// TwinCAT 3 PLC project PLC
// Title: PSAT Nell1
// Company: RMTH GmbH
// ProjectVersion: 0.1
// ProgramVersion: 3.1.4026.20
// libraries:
//   Balluff Sesnor Library TC3, * (Balluff GmbH)
//   IO Link Device Read Conditionmonitoring Data, * (Balluff GmbH)
//   IO Link Device Parametrization , * (Balluff GmbH)
//   RMTH TC3 Library, * (RMTH GmbH)
//   Tc2_ControllerToolbox, * (Beckhoff Automation GmbH)
//   Tc2_Drive, * (Beckhoff Automation GmbH)
//   Tc2_EtherCAT, * (Beckhoff Automation GmbH)
//   Tc2_IoFunctions, * (Beckhoff Automation GmbH)
//   Tc2_Math, * (Beckhoff Automation GmbH)
//   Tc2_MC2, * (Beckhoff Automation GmbH)
//   Tc2_MC2_Drive, * (Beckhoff Automation GmbH)
//   Tc2_Standard, * (Beckhoff Automation GmbH)
//   Tc2_System, * (Beckhoff Automation GmbH)
//   Tc2_TempController, * (Beckhoff Automation GmbH)
//   Tc2_Utilities, * (Beckhoff Automation GmbH)
//   Tc3_EventLogger, * (Beckhoff Automation GmbH)
//   Tc3_Module, * (Beckhoff Automation GmbH)
//   VisuDialogs, * (System)
// project tree:
//   Background/UnitTest/Enumerations/ E_TestCaseState.TcDUT, E_TestResult.TcDUT
//   Background/UnitTest/Interfaces/ ITestCase.TcIO
//   Background/UnitTest/ P_UnitTest.TcPOU
//   Background/UnitTest/TestCases/Base/ FB_TestCaseBase.TcPOU
//   Background/UnitTest/TestCases/ FB_TestCase01FileLog.TcPOU, FB_TestCase02SystemInfo.TcPOU, FB_TestCase03Station.TcPOU
//   Background/UnitTest/TestCases/StationTest/ FB_TestStation.TcPOU
//   Background/UnitTest/TestCases/StationTest/Structures/ ST_TestStation_IN.TcDUT, ST_TestStation_IO.TcDUT, ST_TestStation_OUT.TcDUT
//   DUTs/Configuration/ ST_Configuration.TcDUT
//   GVLs/ CONST.TcGVL, GVL.TcGVL, HMI.TcGVL, IO.TcGVL, NcIO.TcGVL, Safety.TcGVL, Services.TcGVL, Plant.TcGVL
//   / PlcTask.TcTTO, PlcTaskFast.TcTTO
//   POUs/Components/AxisDriver/Enumerations/ E_Axis.TcDUT, E_GearMode.TcDUT, E_JogDirection.TcDUT, E_ManualMode.TcDUT, E_MotionCommand.TcDUT, E_Mover_XTS.TcDUT, E_SoECommand.TcDUT
//   POUs/Components/AxisDriver/ FB_AxisCoupleSync2.TcPOU, FB_AxisDriver.TcPOU, FB_Axis_Ui.TcPOU
//   POUs/Components/AxisDriver/Interfaces/ ITFMotionComponent.TcIO
//   POUs/Components/AxisDriver/Structures/AdditionalAxisIO/ ST_AxisIn.TcDUT, ST_AxisIO.TcDUT, ST_AxisOut.TcDUT, ST_AxisVirtualIO.TcDUT
//   POUs/Components/AxisDriver/Structures/SoE/ ST_AxisSoE.TcDUT
//   POUs/Components/AxisDriver/Structures/ ST_AxisDriverParameter.TcDUT, ST_AxisGearInParameter.TcDUT, ST_AxisGearOutParameter.TcDUT, ST_AxisManager.TcDUT, ST_AxisTorqCtrlParameter.TcDUT, ST_AxisGeneralParameter.TcDUT, ST_AxisHaltParameter.TcDUT, ST_AxisHomingParameter.TcDUT, ST_AxisJogAccParameter.TcDUT, ST_AxisJogParameter.TcDUT, ST_AxisMoveAbsParameter.TcDUT, ST_AxisMoveAddParameter.TcDUT, ST_AxisMoveModParameter.TcDUT, ST_AxisMoveParameter.TcDUT, ST_AxisMoveRelParameter.TcDUT, ST_AxisMoveVelParameter.TcDUT, ST_AxisSetPosParameter.TcDUT, ST_AxisStopParameter.TcDUT, ST_HmiAxisManager.TcDUT
//   POUs/Components/AxisDriver/Utilities/ FB_AxisDistanceTrigger.TcPOU, FB_LimitSwitchRefSim.TcPOU, F_SpeedReached.TcPOU, F_SpeedWindowReached.TcPOU, F_TargetReached.TcPOU, F_TargetReachedOrHigher.TcPOU, F_TargetReachedOrLower.TcPOU, F_TargetWindowReached.TcPOU, F_TargetWindowReachedAxisRef.TcPOU
//   POUs/Components/CylinderDriver/ FB_Cylinder_Ui.TcPOU
//   POUs/Components/Device/ FB_Device.TcPOU, FB_Device_Ui.TcPOU
//   POUs/Components/Device/Structures/ ST_DeviceIn.TcDUT, ST_DeviceIO.TcDUT, ST_DeviceOut.TcDUT
//   POUs/Components/DriveFu/ FB_Drive.TcPOU, FB_Drive_Ui.TcPOU, FB_DriveFuAx_Ui.TcPOU
//   POUs/Components/FurnaceDriver/Enumeration/ E_FurnaceSeq.TcDUT, E_HeatingState.TcDUT
//   POUs/Components/FurnaceDriver/ FB_FurnaceDriver.TcPOU
//   POUs/Components/FurnaceDriver/Structures/ ST_FurnaceIn.TcDUT, ST_FurnaceIO.TcDUT, ST_FurnaceOut.TcDUT
//   POUs/Components/_Base/ FB_ComponentBase.TcPOU, FB_ManualUiBase.TcPOU
//   POUs/Components/_Base/Interfaces/ I_ManualUi.TcIO, ITFComponent.TcIO
//   POUs/Components/_Enumerations/ E_ComponentState.TcDUT, E_Component.TcDUT, E_ComponentType.TcDUT
//   POUs/Components/_Structures/ ST_Coordinate.TcDUT, ST_Curve.TcDUT, ST_Point.TcDUT, ST_3DPoint.TcDUT
//   POUs/HMI/Events/ FB_EventHandler.TcPOU
//   POUs/HMI/Events/Interfaces/ I_EventHandler.TcIO
//   POUs/HMI/Provider/HwHmi/ FB_HMI_PROVIDER_HW.TcPOU
//   POUs/HMI/Provider/HwHmi/Structures/+P10A_Pult/ ST_P10A_Pult_IN.TcDUT, ST_P10A_Pult_OUT.TcDUT
//   POUs/HMI/Provider/HwHmi/Structures/+P50A_Haupt/ ST_P50A_Haupt_IN.TcDUT, ST_P50A_Haupt_OUT.TcDUT
//   POUs/HMI/Provider/HwHmi/Structures/+P51A_EuchnerHandBedien/ ST_P51A_EuchnerHandB_IN.TcDUT, ST_P51A_EuchnerHandB_OUT.TcDUT
//   POUs/HMI/Provider/HwHmi/Structures/ HMI_PROVIDER_HW_IN.TcDUT, HMI_PROVIDER_HW_OUT.TcDUT, HMI_PROVIDER_HW_IO.TcDUT
//   POUs/HMI/Provider/HwHmi/Structures/_Base/ ST_PxAB_SxHandAsBs_IN.TcDUT, ST_PxAB_SxHandAsBs_OUT.TcDUT
//   POUs/HMI/Provider/Tc3Hmi/ FB_HMI_Provider_TC3.TcPOU
//   POUs/HMI/Provider/Tc3Hmi/Structures/Stations/ ST_StationToTc3Hmi.TcDUT, ST_StationFromTc3Hmi.TcDUT
//   POUs/HMI/Provider/Tc3Hmi/Structures/ ST_FromTc3Hmi.TcDUT, ST_Header.TcDUT, ST_HMI_Tc3.TcDUT, ST_ToTc3Hmi.TcDUT, ST_ToTc3HmiConditionMonitoring.TcDUT, ST_ToTc3Hmi_Door.TcDUT, ST_ToTc3Hmi_EmergencyStop.TcDUT
//   POUs/HMI/Provider/Tc3Hmi/Structures/UserControls/DataGrid/ ST_UserControlGrid_FromHmi.TcDUT, ST_UserControlGrid_ToHmi.TcDUT
//   POUs/HMI/Provider/Tc3Hmi/Structures/UserControls/ManualControl Axis/ ST_UserControl_Manual_Axis_FromHmi.TcDUT, ST_UserControl_Manual_Axis_Item.TcDUT, ST_UserControl_Manual_Axis_Item_String.TcDUT, ST_UserControl_Manual_Axis_ToHmi.TcDUT
//   POUs/HMI/Provider/Tc3Hmi/Structures/UserControls/ManualControl Cylinder/ ST_UserControl_Manual_Cylinder_FromHmi.TcDUT, ST_UserControl_Manual_Cylinder_ToHmi.TcDUT
//   POUs/HMI/Provider/Tc3Hmi/Structures/UserControls/ManualControl Device/ ST_UserControl_Manual_Device_FromHmi.TcDUT, ST_UserControl_Manual_Device_ToHmi.TcDUT
//   POUs/HMI/Provider/Tc3Hmi/Structures/UserControls/ManualControl Drive/ ST_UserControl_Manual_Drive_FromHmi.TcDUT, ST_UserControl_Manual_Drive_ToHmi.TcDUT
//   POUs/HMI/Provider/Tc3Hmi/Structures/UserControls/SensorActor/ ST_ToVisuSensorActor.TcDUT
//   POUs/HMI/Provider/_Base/ FB_HMI_PROVIDER_BASE.TcPOU
//   POUs/HMI/Provider/_Enumerations/ E_HMI_CONTROL_REQUEST.TcDUT, E_HMI_PROVIDER.TcDUT
//   POUs/HMI/Provider/_Interfaces/ ITF_HMI_PROVIDER.TcIO
//   POUs/HMI/Utilities/DynTxt/ F_CreateDynText.TcPOU, F_CreateDynTextDefault.TcPOU, F_CreateDynTextDefaultS.TcPOU, F_CreateDynTextEx.TcPOU
//   POUs/HMI/Utilities/ FB_CounterHandling.TcPOU, FB_MonitoringHandling.TcPOU, FB_ProviderRequestTrigger.TcPOU, F_AlarmPrioToText.TcPOU, F_AlarmPrioToHexColor.TcPOU, FB_HmiBaseControlTrigger.TcPOU
//   POUs/HMI/Utilities/SettingsHandling/ FB_SettingsHandling.TcPOU, F_SettingItemHandling.TcPOU, F_SettingItemHandlingB.TcPOU, F_SettingItemHandlingF.TcPOU, F_SettingItemHandlingI.TcPOU, F_SettingItemHandlingWs.TcPOU
//   POUs/HMI/Utilities/Tracking/ F_TrackSettingChangesB.TcPOU, F_TrackSettingChangesF.TcPOU, F_TrackSettingChangesI.TcPOU, F_TrackSettingChangesT.TcPOU, F_TrackSettingChangesWs.TcPOU
//   POUs/HMI/Utilities/Validation/ F_ChkSettingLimit.TcPOU, F_ChkSettingLimitF.TcPOU, F_ChkSettingLimitN.TcPOU, F_ChkSettingUserLevel.TcPOU
//   POUs/HMI/ P_HMI_Controller.TcPOU
//   POUs/HMI/_Enumerations/ E_Axis_JogMode.TcTLEO, E_DataType.TcTLEO, E_Drive_JogMode.TcDUT, E_Language.TcDUT, E_ManualObjectControlMode.TcDUT, E_Popup.TcDUT, E_RecipeMode.TcTLEO, E_User.TcTLEO, E_User_Level.TcDUT
//   POUs/HMI/_Structures/Counter/ E_CounterReaction.TcTLEO, ST_CounterControlIn.TcDUT, ST_CounterControlOut.TcDUT, ST_Counter_Item_String.TcDUT
//   POUs/HMI/_Structures/Data/ ST_Data_Item_String.TcDUT, ST_Data_Item.TcDUT
//   POUs/HMI/_Structures/Monitoring/ ST_GridObject_Name_Value1_Event1_Value2_Event2_Unit.TcDUT, ST_GridObject_Name_sValue_Unit.TcDUT, ST_Monitoring_Station.TcDUT, ST_Monitoring.TcDUT, ST_Monitoring_Base.TcDUT, ST_Monitoring_Module.TcDUT
//   POUs/HMI/_Structures/Popup/ E_PopupSymbol.TcDUT, ST_PopUp_FromHmi.TcDUT, ST_PopUp_ToHmi.TcDUT
//   POUs/HMI/_Structures/Recipe/ ST_HMI_RECIPE_IN.TcDUT, ST_HMI_RECIPE_OUT.TcDUT
//   POUs/HMI/_Structures/Safety/ ST_HMI_SAFETY_IN.TcDUT, ST_HMI_SAFETY_OUT.TcDUT
//   POUs/HMI/_Structures/Settngs/ ST_HMI_CONTROL_SETTING_IN.TcDUT, ST_HMI_CONTROL_SETTING_OUT.TcDUT, ST_HMI_CONTROL_SETTING_STATION_OUT.TcDUT, ST_HMI_CONTROL_SETTING_MODULE_OUT.TcDUT, ST_HMI_CONTROL_SETTING_ITEM_IN.TcDUT, ST_HMI_CONTROL_SETTING_ITEM_OUT.TcDUT
//   POUs/HMI/_Structures/SetupPlant/ E_SetupPlantShape.TcDUT, E_SetupPlantStateShape.TcDUT, ST_SetupPlant_Item_String.TcDUT
//   POUs/HMI/_Structures/ ST_HMI.TcDUT, ST_HMI_IN.TcDUT, ST_HMI_InOut.TcDUT, ST_HMI_OUT.TcDUT, ST_NameValue.TcDUT
//   POUs/HMI/_Structures/UserManagment/ ST_HMI_USER_MGMT_IN.TcDUT, ST_HMI_USER_MGMT_OUT.TcDUT, ST_User_Management.TcDUT
//   POUs/HMI/_Structures/_Base/Button/ ST_HMI_BUTTON_IN.TcDUT, ST_HMI_BUTTON_OUT.TcDUT
//   POUs/HMI/_Structures/_Base/Common/ ST_HMI_BASE_CONTROL_IN.TcDUT, ST_HMI_BASE_CONTROL_OUT.TcDUT, ST_HMI_BASE_SPECIAL_IN.TcDUT, ST_HMI_GRID_IN.TcDUT, ST_HMI_NAME_VALUE_STRING.TcDUT, ST_HMI_TRAFFIC_LIGHT_OUT.TcDUT
//   POUs/HMI/_Structures/_Base/Manual/ManualControl Axis/ ST_HMI_MANUAL_AXIS_IN.TcDUT, ST_HMI_MANUAL_AXIS_ITEM.TcDUT, ST_HMI_MANUAL_AXIS_ITEM_STRING.TcDUT, ST_HMI_MANUAL_AXIS_OUT.TcDUT
//   POUs/HMI/_Structures/_Base/Manual/ManualControl Cylinder/ ST_HMI_MANUAL_CYLINDER_IN.TcDUT, ST_HMI_MANUAL_CYLINDER_OUT.TcDUT
//   POUs/HMI/_Structures/_Base/Manual/ManualControl Device/ ST_HMI_MANUAL_DEVICE_IN.TcDUT, ST_HMI_MANUAL_DEVICE_OUT.TcDUT
//   POUs/HMI/_Structures/_Base/Manual/ManualControl Drive/ ST_HMI_MANUAL_DRIVE_IN.TcDUT, ST_HMI_MANUAL_DRIVE_OUT.TcDUT
//   POUs/HMI/_Structures/_Base/Module/ ST_HMI_BASE_MODULE_IN.TcDUT, ST_HMI_BASE_MODULE_MANUAL_IN.TcDUT, ST_HMI_BASE_MODULE_MANUAL_OUT.TcDUT, ST_HMI_BASE_MODULE_OUT.TcDUT
//   POUs/HMI/_Structures/_Base/Station/ ST_HMI_BASE_STATION_IN.TcDUT, ST_HMI_BASE_STATION_MANUAL_IN.TcDUT, ST_HMI_BASE_STATION_MANUAL_OUT.TcDUT, ST_HMI_BASE_STATION_OUT.TcDUT
//   POUs/HMI/_Structures/_Base/ ST_HMI_BASE_IN.TcDUT, ST_HMI_BASE_OUT.TcDUT
//   POUs/HMI/_Structures/_Common/ ST_HexColor.TcDUT, ST_HMI_COLOR_STRING.TcDUT, ST_Text.TcDUT, ST_DefaultHmiToPlc.TcDUT
//   POUs/HMI/_Structures/_TextLists/ ST_Text_List_Components.TcDUT, ST_Text_List_Global.TcDUT, ST_Text_List_Safety.TcDUT, ST_Text_List_System.TcDUT
//   POUs/Items/TcaCarrier/Enumerations/ eTcaCarrierCmd.TcDUT, eTcaCarrierLayout.TcDUT
//   POUs/Items/TcaCarrier/Structures/ TcaCarrierConfig.TcDUT, TcaCarrierData.TcDUT, TcaCarrierService.TcDUT
//   POUs/Items/TcaCarrier/ TcaCarrier.TcPOU
//   POUs/Items/TcaTrolley/Structures/ TcaTrolleyConfig.TcDUT, TcaTrolleyData.TcDUT, TcaTrolleyService.TcDUT
//   POUs/Items/TcaTrolley/ TcaTrolley.TcPOU
//   POUs/Items/TcaWorkpiece/Enumerations/ eTcaWorkpieceShape.TcDUT, eTcaWorkpieceStatus.TcDUT
//   POUs/Items/TcaWorkpiece/Structures/ TcaWorkpieceData.TcDUT
//   POUs/Items/TcaWorkpiece/ TcaWorkpieceControl.TcPOU
//   POUs/ MAIN.TcPOU, MAIN_Fast.TcPOU
//   POUs/Plant/_Enumerations/ E_Module.TcDUT, E_PlantSettings.TcDUT, E_ProductionSettings.TcDUT, E_ProductSettings.TcDUT, E_Station.TcDUT
//   POUs/Plant/M001_Module/_Enumerations/ E_M001_Settings.TcDUT
//   POUs/Plant/M001_Module/_Structures/ ST_M001_HMI_IN.TcDUT, ST_M001_Interface.TcDUT, ST_M001_HMI_OUT.TcDUT, ST_M001_IO.TcDUT, ST_M001_IO_IN.TcDUT, ST_M001_IO_OUT.TcDUT
//   POUs/Plant/ P_Plant.TcPOU
//   POUs/Plant/ST010_OvenA/_Structures/ ST_St010_HMI_IN.TcDUT, ST_St010_Interface.TcDUT, ST_St010_HMI_IN_OUT.TcDUT, ST_St010_HMI_OUT.TcDUT, ST_St010_IO_IN.TcDUT, ST_St010_IO.TcDUT, ST_St010_IO_OUT.TcDUT
//   POUs/Plant/ST020_OvenB/_Enumerations/ E_St020_Settings.TcDUT
//   POUs/Plant/ST020_OvenB/ FB_St020_OvenB.TcPOU
//   POUs/Plant/ST020_OvenB/_Structures/ ST_St020_HMI_IN_OUT.TcDUT, ST_St020_HMI_IN.TcDUT, ST_St020_Interface.TcDUT, ST_St020_IO.TcDUT, ST_St020_IO_IN.TcDUT, ST_St020_IO_OUT.TcDUT, ST_St020_HMI_OUT.TcDUT
//   POUs/Plant/ST030_Handling/_Enumerations/ E_St030_Command.TcDUT, E_St030_EmptySlotChk.TcDUT, E_St030_Settings.TcDUT
//   POUs/Plant/ST030_Handling/ FB_St030_Handling.TcPOU
//   POUs/Plant/ST030_Handling/_Structures/ ST_St030_HMI_OUT.TcDUT, ST_St030_HMI_IN.TcDUT, ST_St030_Interface.TcDUT, ST_St030_Command.TcDUT, ST_St030_IO.TcDUT, ST_St030_IO_IN.TcDUT, ST_St030_IO_OUT.TcDUT, ST_St030_HMI_IN_OUT.TcDUT, ST_XZ_Point.TcDUT
//   POUs/Plant/ST040_Storage/_Enumerations/ E_St040_Settings.TcDUT
//   POUs/Plant/ST040_Storage/ FB_St040_Storage.TcPOU
//   POUs/Plant/ST040_Storage/_Structures/ ST_St040_HMI_IN.TcDUT, ST_St040_HMI_IN_OUT.TcDUT, ST_St040_HMI_OUT.TcDUT, ST_St040_IO.TcDUT, ST_St040_IO_IN.TcDUT, ST_St040_IO_OUT.TcDUT, ST_St040_Interface.TcDUT
//   POUs/Plant/ST050_Mould/_Enumerations/ E_St050_Settings.TcDUT
//   POUs/Plant/ST050_Mould/ FB_St050_Mould.TcPOU
//   POUs/Plant/ST050_Mould/_Structures/ ST_St050_Interface.TcDUT, ST_St050_IO.TcDUT, ST_St050_IO_IN.TcDUT, ST_St050_IO_OUT.TcDUT, TcaEngelCastingCarrierInput.TcDUT, TcaEngelCastingCarrierJob.TcDUT, TcaEngelCastingCarrierJobStatus.TcDUT, TcaEngelCastingCarrierOutput.TcDUT, TcaEngelCastingCarrierStatus.TcDUT
//   POUs/Plant/_Base/Interfaces/ IModule.TcIO, IStation.TcIO
//   POUs/Plant/_Specific/Components/TcaWorkpiece/ TcaWorkpieceControl.TcPOU (not stored)
//   POUs/Plant/_Specific/S01_Workpiece/Enumerations/ E_HMI_WP_CMD.TcDUT (not stored), E_ProcessState.TcDUT (not stored), E_ProcessStep.TcDUT (not stored)
//   POUs/Plant/_Specific/S01_Workpiece/ FB_Workpiece.TcPOU (not stored), FB_WorkpieceRef.TcPOU (not stored)
//   POUs/Plant/_Specific/S01_Workpiece/Structures/ ST_HMI_WP_CMD.TcDUT (not stored), ST_Workpiece.TcDUT (not stored)
//   POUs/Plant/_Specific/S02_Pallet/Enumerations/ E_HMI_PL_CMD.TcDUT (not stored)
//   POUs/Plant/_Specific/S02_Pallet/ FB_Pallet.TcPOU (not stored), FB_PalletRef.TcPOU (not stored)
//   POUs/Plant/_Specific/S02_Pallet/Structures/ ST_HMI_PL_CMD.TcDUT (not stored), ST_Pallet.TcDUT (not stored)
//   POUs/Plant/_Specific/S03_Trolley/Enumerations/ E_HMI_TR_CMD.TcDUT (not stored)
//   POUs/Plant/_Specific/S03_Trolley/ FB_Trolley.TcPOU (not stored)
//   POUs/Plant/_Specific/S03_Trolley/Structures/ ST_HMI_TR_CMD.TcDUT (not stored), ST_Trolley.TcDUT (not stored)
//   POUs/Plant/_Structures/ControlCabinet/ ST_ControlCabinetIn.TcDUT, ST_ControlCabinetIO.TcDUT, ST_ControlCabinetOut.TcDUT
//   POUs/Plant/_Structures/Counter/ ST_Counter.TcDUT
//   POUs/Plant/_Structures/Objects/ ST_Objects.TcDUT, ST_Object_Item.TcDUT
//   POUs/Plant/_Structures/Settings/ ST_ModuleDynSettings.TcDUT, ST_Settings.TcDUT, ST_StationDynSettings.TcDUT
//   POUs/Plant/_Structures/ ST_DefaultEventClasses.TcDUT, ST_MODULE_STATIONS_INFO.TcDUT, ST_MODULES_INFO.TcDUT
//   POUs/Safety/Components/Euchner_MBM/ FB_Euchner_MBM.TcPOU
//   POUs/Safety/Components/Euchner_MBM/Structure/ ST_Euchner_MBM_HW_IN.TcDUT, ST_Euchner_MBM_HW_OUT.TcDUT, ST_Euchner_MBM_IN.TcDUT, ST_Euchner_MBM_OUT.TcDUT, ST_MBM_IO.TcDUT
//   POUs/Safety/Components/Euchner_MGB2/ FB_SafeDoorMGB2.TcPOU
//   POUs/Safety/Components/Euchner_MGB2/Structure/MGB2/ ST_Euchner_MGB2_HW_IN.TcDUT, ST_Euchner_MGB2_HW_OUT.TcDUT, ST_Euchner_MGB2_IN.TcDUT, ST_Euchner_MGB2_OUT.TcDUT
//   POUs/Safety/Components/Euchner_MGB2/Structure/MSM/ ST_Euchner_MSM_DA_IN.TcDUT, ST_Euchner_MSM_DA_OUT.TcDUT, ST_Euchner_MSM_HW_IN.TcDUT, ST_Euchner_MSM_HW_OUT.TcDUT, ST_Euchner_MSM_IN.TcDUT, ST_Euchner_MSM_OUT.TcDUT
//   POUs/Safety/Components/Euchner_MGB2/Structure/ ST_MGB2_IO.TcDUT
//   POUs/Safety/Components/SafetyDoor/ FB_SafetyDoor.TcPOU
//   POUs/Safety/Components/SafetyDoor/Structure/ ST_SafetyDoor_IN.TcDUT, ST_SafetyDoor_IO.TcDUT, ST_SafetyDoor_OUT.TcDUT
//   POUs/Safety/Enumerations/ E_EDM_Out.TcDUT, E_Safety_Actor.TcDUT, E_EmergencyStop.TcDUT, E_Door.TcDUT
//   POUs/Safety/ P_Safety.TcPOU
//   POUs/Safety/Structures/Diag/ E_HistoryDiagDevices.TcDUT, ST_DiagHistory.TcDUT, ST_DiagMessage.TcDUT, ST_DiagMessageFlags.TcDUT, ST_ELM3xxxPAIInfoData.TcDUT, ST_MessageItem.TcDUT, ST_SafetyDiagInfo.TcDUT
//   POUs/Safety/Structures/ ST_SafetyIn.TcDUT, ST_SafetyIO.TcDUT, ST_SafetyOut.TcDUT
//   POUs/Safety/TwinSAFE_Diagnose/ FB_Diagnosis_History.TcPOU, FB_TwinSAFEDiag_EDM.TcPOU, FB_TwinSAFEDiag_EmergencyStop.TcPOU, FB_TwinSAFEDiag_MachineMonitoring.TcPOU, FB_TwinSAFEDiag_TwoHand.TcPOU, FB_TwinSAFE_HW_Diag.TcPOU
//   POUs/Plant/M001_Module/ FB_M001_Module.TcPOU
//   POUs/Plant/ST010_OvenA/_Enumerations/ E_St010_Settings.TcDUT
//   POUs/Plant/_Base/ FB_ModuleBase.TcPOU, FB_StationBase.TcPOU
//   POUs/Plant/ST010_OvenA/ FB_St010_OvenA.TcPOU
//   POUs/System/ P_SysSrv.TcPOU
//   POUs/System/Recipe/ FB_RecipeManager.TcPOU
//   POUs/System/Supervision/Enumerations/Alarmsystem/ E_AlarmPriority.TcDUT, E_AlarmState.TcDUT, E_EventReaction.TcDUT
//   POUs/System/Supervision/Enumerations/ E_EtherCatBox.TcDUT
//   POUs/System/Supervision/EtherCAT/Enumerations/ E_EcDeviceState.TcDUT
//   POUs/System/Supervision/EtherCAT/ FB_DiagEtherCAT.TcPOU
//   POUs/System/Supervision/ImplicitChecks/ CheckBounds.TcPOU, CheckDivDInt.TcPOU, CheckDivLInt.TcPOU, CheckDivLReal.TcPOU, CheckDivReal.TcPOU, CheckPointer.TcPOU, CheckRangeSigned.TcPOU, CheckRangeUnsigned.TcPOU
//   POUs/System/Supervision/ P_Supervision.TcPOU
//   POUs/System/Supervision/Structures/ ST_EcMaster_In.TcDUT, ST_GridObject_Register.TcDUT, ST_SystemVars.TcDUT
//   POUs/System/Utilities/Convert/ F_DegPerSecToDegPerMin.TcPOU, F_DegPerSecToUpm.TcPOU, F_Diagnostic_EcDeviceState.TcPOU, F_Diagnostic_EcLinkState.TcPOU, F_Diagnostic_EcMasterDeviceState.TcPOU, F_EcDeviceTimeStampToTime.TcPOU, F_MeterPerMinToMmPerSec.TcPOU, F_MmPerSecToMmPerMin.TcPOU, F_UpmToDegreePerSec.TcPOU, F_MmPerMinToMmPerSec.TcPOU, F_MmPerSecToMeterPerMin.TcPOU, F_DegPerMinToDegPerSec.TcPOU
//   POUs/System/Utilities/Counter/ E_Counter.TcDUT, E_CounterMode.TcDUT, F_Counter.TcPOU, ST_Counter_Item.TcDUT
//   POUs/System/Utilities/CSV/ FB_WriteCSV.TcPOU
//   POUs/System/Utilities/CSV/Structures/ ST_FillOrder.TcDUT
//   POUs/System/Utilities/ FB_JogTrigTon.TcPOU, FB_Puls_On_Off.TcPOU, FB_RtrigFtrigTof.TcPOU, FB_RtrigFtrig.TcPOU, FB_StableValue.TcPOU, FB_ToggleSwitch.TcPOU
//   POUs/System/Utilities/Functions/ F_ADD_REF_F.TcPOU, F_AND_REF_EX.TcPOU, F_Byte_To_DWord.TcPOU, F_Byte_To_Word.TcPOU, F_ColorToStringHexColor.TcPOU, F_CutInstancePath.TcPOU, F_FindBackupItem.TcPOU, F_FormatString.TcPOU, F_InitDynDataItem.TcPOU, F_InRange.TcPOU, F_Log_Add.TcPOU, F_OR_REF.TcPOU, F_AND_REF.TcPOU, F_OR_REF_EX.TcPOU, F_Real_To_Byte.TcPOU, F_RestoreSettingValues.TcPOU, F_Settings_Management.TcPOU, F_Settings_Row_Delete.TcPOU, F_Settings_Row_Insert.TcPOU, F_Trend.TcPOU, F_CopyDataItemValues.TcPOU
//   POUs/System/Utilities/Interfaces/ I_StringBuilder.TcIO, I_WStringBuilder.TcIO
//   POUs/System/Utilities/Sequencer/ FB_SequenceHelper.TcPOU, FB_SequenceHelperSb.TcPOU
//   POUs/System/Utilities/String/ FB_StringBuilder.TcPOU, FB_WStringBuilder.TcPOU, F_Replace.TcPOU, WConcat10.TcPOU, WConcat2x.TcPOU, WConcat3.TcPOU, WConcat4.TcPOU, WConcat5.TcPOU, WConcat6.TcPOU, WConcat7.TcPOU, WConcat8.TcPOU, WConcat9.TcPOU
//   POUs/System/Utilities/Var2File/ FB_Var2File.TcPOU
//   POUs/System/Utilities/Var2File/Structures/ ST_Var2File_Com.TcDUT, ST_Var2File_Config.TcDUT
// real-time tasks:
//   TASK PlcTask: cycle T#5ms, priority 10, ADS port 350
//   TASK PlcTaskFast: cycle T#1ms, priority 4, ADS port 351
// motion (NC):
//   TASK NC-Task 1 SAF: cycle T#2ms, priority 6, ADS port 501
//   TASK NC-Task 1 SVB: cycle T#10ms, priority 12, ADS port 511
//   AXIS Oven B CH1 (id 14)
//     Dynamic: Acceleration=282800000, Deceleration=282800000, Jerk=2.85628e+17
//     Velo: RefSearch=25, RefSync=25, SlowManual=14, FastManual=28, Maximum=28
//     PositionAreaControl: Enable=false
//     TargetPosControl: Enable=false
//     OtherSettings: AllowMotionCmdToSlave=true
//     encoder EncType=7
//       EncPara: ScaleFactorNumerator=0.001879, Offset=-1.4, MaxCount=#x0000ffff, ReferenceSystem=1
//     drive DrvType=23
//       Analog: VeloReferenz=28, TorqueSetpointScale=10, ScaleFactorActTorque=0.1
//       TimeComp: TaskDelayCycles=1
//     controller CtrType=1
//       CtrPara: PriorControlFactor=1
//         PosDiffControl: Enable=false
//         Observer: BandWidth=20
//   AXIS Oven B CH2 (id 15)
//     Dynamic: Acceleration=282800000, Deceleration=282800000, Jerk=2.85628e+17
//     Velo: RefSearch=25, RefSync=25, SlowManual=14, FastManual=28, Maximum=28
//     PositionAreaControl: Enable=false
//     TargetPosControl: Enable=false
//     OtherSettings: AllowMotionCmdToSlave=true
//     encoder EncType=7
//       EncPara: ScaleFactorNumerator=0.001879, Offset=-1.4, MaxCount=#x0000ffff, ReferenceSystem=1
//     drive DrvType=23
//       Analog: VeloReferenz=28, TorqueSetpointScale=10, ScaleFactorActTorque=0.1
//       TimeComp: TaskDelayCycles=1
//     controller CtrType=1
//       CtrPara: PriorControlFactor=1
//         PosDiffControl: Enable=false
//         Observer: BandWidth=20
//   AXIS Rackfeeder X (id 16)
//     Dynamic: AccelerationMaximum=5000, DecelerationMaximum=5000, Acceleration=2150.09, Deceleration=2150.09, Jerk=9085.86
//     Velo: RefSearch=16.41285, RefSync=16.41285, SlowManual=10, FastManual=60, Fast=1641.285, Maximum=1641.29
//     OtherSettings: AllowMotionCmdToSlave=true
//     encoder EncType=8
//       EncPara: ScaleFactorNumerator=150, ScaleFactorDenominator=10485760, MaxCount=#xffffffff, EncPositionSource=1
//     drive DrvType=9
//       DrvPara: MaxCount=#xffffffff, DriveControlDWord=#x00030100
//         Analog: VeloReferenz=1805.4135, VeloScale=1.02400649589962, TorqueSetpointScale=10, ScaleFactorActTorque=0.1
//         TimeComp: TaskDelayCycles=1
//     controller CtrType=1
//       CtrPara: PriorControlFactor=1
//         Observer: BandWidth=20
//   AXIS Rackfeeder Y (id 17)
//     Dynamic: Acceleration=2004.51, Deceleration=2004.51, Jerk=8036.12
//     Velo: RefSearch=15.04511, RefSync=15.04511, SlowManual=10, FastManual=60, Fast=1504.511, Maximum=1504.51
//     OtherSettings: AllowMotionCmdToSlave=true
//     encoder EncType=8
//       EncPara: ScaleFactorNumerator=220, ScaleFactorDenominator=16777216, MaxCount=#xffffffff, EncPositionSource=1
//     drive DrvType=9
//       DrvPara: MaxCount=#xffffffff, DriveControlDWord=#x00030100
//         Analog: VeloReferenz=1654.9621, VeloScale=1.02400649589962, TorqueSetpointScale=10, ScaleFactorActTorque=0.1
//         TimeComp: TaskDelayCycles=1
//     controller CtrType=1
//       CtrPara: PriorControlFactor=1
//         Observer: BandWidth=20
//   AXIS Rackfeeder Z (id 18)
//     Dynamic: Acceleration=500, Deceleration=500, Jerk=500
//     Velo: RefSearch=30.19555, RefSync=30.19555, SlowManual=35, FastManual=210, Fast=3019.555, Maximum=3019.555
//     OtherSettings: AllowMotionCmdToSlave=true
//     encoder EncType=8
//       EncPara: ScaleFactorNumerator=27.59625, ScaleFactorDenominator=1048576, MaxCount=#xffffffff, EncPositionSource=1
//     drive DrvType=9
//       DrvPara: MaxCount=#xffffffff, DriveControlDWord=#x00030100
//         Analog: VeloReferenz=3321.5105, VeloScale=1.02400649589962, TorqueSetpointScale=10, ScaleFactorActTorque=0.1
//         TimeComp: TaskDelayCycles=1
//     controller CtrType=1
//       CtrPara: PriorControlFactor=1
//         Observer: BandWidth=20
//   AXIS Oven B (id 21)
//     Dynamic: Acceleration=1231.0125, Deceleration=1231.0125, Jerk=3693.0375
//     Velo: RefSearch=8.20675, RefSync=8.20675, SlowManual=20, FastManual=120, Fast=820.675, Maximum=820.675
//     OtherSettings: AllowMotionCmdToSlave=true
//     encoder EncType=8
//       EncPara: ScaleFactorNumerator=120, ScaleFactorDenominator=16777216, Inverse=true, MaxCount=#xffffffff, EncPositionSource=1
//     drive DrvType=9
//       DrvPara: Inverse=true, MaxCount=#xffffffff, DriveControlDWord=#x00030100
//         Analog: VeloReferenz=902.7425, VeloScale=1.02400649589962, TorqueSetpointScale=10, ScaleFactorActTorque=0.1
//         TimeComp: TaskDelayCycles=1
//     controller CtrType=1
//       CtrPara: PriorControlFactor=1
//         Observer: BandWidth=20
//   AXIS Oven A (id 20)
//     Dynamic: Acceleration=1231.01, Deceleration=1231.01, Jerk=3693.04
//     Velo: RefSearch=8.20675, RefSync=8.20675, SlowManual=20, FastManual=120, Fast=820.675, Maximum=820.675
//     OtherSettings: AllowMotionCmdToSlave=true
//     encoder EncType=8
//       EncPara: ScaleFactorNumerator=120, ScaleFactorDenominator=16777216, Inverse=true, MaxCount=#xffffffff, EncPositionSource=1
//     drive DrvType=9
//       DrvPara: Inverse=true, MaxCount=#xffffffff, DriveControlDWord=#x00030100
//         Analog: VeloReferenz=902.7425, VeloScale=1.02400649589962, TorqueSetpointScale=10, ScaleFactorActTorque=0.1
//         TimeComp: TaskDelayCycles=1
//     controller CtrType=1
//       CtrPara: PriorControlFactor=1
//         Observer: BandWidth=20
//   AXIS Oven A CH1 (id 1)
//     Dynamic: Acceleration=282800000, Deceleration=282800000, Jerk=2.85628e+17, DelayTime=0.01, OverrideType=4
//     Velo: RefSearch=25, RefSync=25, SlowManual=14, FastManual=28, Maximum=28
//     PositionAreaControl: Enable=false
//     TargetPosControl: Enable=false
//     OtherSettings: AllowMotionCmdToSlave=true
//     encoder EncType=7
//       EncPara: ScaleFactorNumerator=0.001879, Offset=-1.4, EncMode=1, MaxCount=#x0000ffff, ReferenceSystem=1
//         FilterTime: TVelo=0.1
//         SoftEndMinControl: Range=-5
//         SoftEndMaxControl: Range=30
//         ActPosCorrection: Enable=true, Time=1
//     drive DrvType=23
//       Analog: VeloReferenz=28, TorqueSetpointScale=10, ScaleFactorActTorque=0.1
//       TimeComp: TaskDelayCycles=1
//     controller CtrType=1
//       CtrPara: PriorControlFactor=1
//         PosDiffControl: Enable=false
//         Observer: BandWidth=20
//   AXIS Oven A CH2 (id 13)
//     Dynamic: Acceleration=282800000, Deceleration=282800000, Jerk=2.85628e+17
//     Velo: RefSearch=25, RefSync=25, SlowManual=14, FastManual=28, Maximum=28
//     PositionAreaControl: Enable=false
//     TargetPosControl: Enable=false
//     OtherSettings: AllowMotionCmdToSlave=true
//     encoder EncType=7
//       EncPara: ScaleFactorNumerator=0.001879, Offset=-1.4, MaxCount=#x0000ffff, ReferenceSystem=1
//     drive DrvType=23
//       Analog: VeloReferenz=28, TorqueSetpointScale=10, ScaleFactorActTorque=0.1
//       TimeComp: TaskDelayCycles=1
//     controller CtrType=1
//       CtrPara: PriorControlFactor=1
//         PosDiffControl: Enable=false
//         Observer: BandWidth=20
//   AXIS Storage A (id 2)
//     Dynamic: Acceleration=282800000, Deceleration=282800000, Jerk=2.85628e+17, DelayTime=0.01, OverrideType=4
//     Velo: RefSearch=25, RefSync=25, SlowManual=14, FastManual=28, Maximum=28
//     PositionAreaControl: Enable=false
//     TargetPosControl: Enable=false
//     OtherSettings: AllowMotionCmdToSlave=true
//     encoder EncType=7
//       EncPara: ScaleFactorNumerator=0.001879, Offset=-1.4, EncMode=1, MaxCount=#x0000ffff, ReferenceSystem=1
//         FilterTime: TVelo=0.1
//         SoftEndMinControl: Range=-5
//         SoftEndMaxControl: Range=30
//         ActPosCorrection: Enable=true, Time=1
//     drive DrvType=23
//       Analog: VeloReferenz=28, TorqueSetpointScale=10, ScaleFactorActTorque=0.1
//       TimeComp: TaskDelayCycles=1
//     controller CtrType=1
//       CtrPara: PriorControlFactor=1
//         PosDiffControl: Enable=false
//         Observer: BandWidth=20
//   AXIS Storage B (id 3)
//     Dynamic: Acceleration=282800000, Deceleration=282800000, Jerk=2.85628e+17
//     Velo: RefSearch=25, RefSync=25, SlowManual=14, FastManual=28, Maximum=28
//     PositionAreaControl: Enable=false
//     TargetPosControl: Enable=false
//     OtherSettings: AllowMotionCmdToSlave=true
//     encoder EncType=7
//       EncPara: ScaleFactorNumerator=0.001879, Offset=-1.4, MaxCount=#x0000ffff, ReferenceSystem=1
//     drive DrvType=23
//       Analog: VeloReferenz=28, TorqueSetpointScale=10, ScaleFactorActTorque=0.1
//       TimeComp: TaskDelayCycles=1
//     controller CtrType=1
//       CtrPara: PriorControlFactor=1
//         PosDiffControl: Enable=false
//         Observer: BandWidth=20
// I/O:
//   DEVICE Gerät 3 (EtherCAT), AmsNetId 172.31.31.4.4.1
//     Klemme 1 (EK1100) [EK1100 EtherCAT-Koppler (2A E-Bus)]
//       Klemme 33 (EL6910) [EL6910, TwinSAFE PLC]
//       Klemme 3 (EL1904) [EL1904, 4 K. Safety Eingang 24V, TwinSAFE]
//         modules: Module 1 (FSOES)
//       Klemme 4 (EL2904) [EL2904, 4 K. Safety Ausgang 24V, 0.5A, TwinSAFE]
//         modules: Module 1 (FSOES), Module 2 (DO)
//       Klemme 5 (EL1104) [EL1104 4K. Dig. Eingang 24V, 3ms, Sensorversorgung]
//       Klemme 6 (EL1104) [EL1104 4K. Dig. Eingang 24V, 3ms, Sensorversorgung]
//       Klemme 7 (EL6224) [EL6224 (IO Link Master)]
//       ENGEL Interface (EL1008) [EL1008 8K. Dig. Eingang 24V, 3ms]
//       ENGEL Interface (EL2624) [EL2624 4K. Relais Ausgang, Schließer (125V AC / 30V DC)]
//       Klemme 43 (EL1904)
//       Ovens (EK1122) [EK1122 2-Port EtherCAT-Abzweig]
//         Oven_A (EK1100) [EK1100 EtherCAT-Koppler (2A E-Bus)]
//           Klemme 10 (EL1904) [EL1904, 4 K. Safety Eingang 24V, TwinSAFE]
//             modules: Module 1 (FSOES)
//           Klemme 11 (EL2904) [EL2904, 4 K. Safety Ausgang 24V, 0.5A, TwinSAFE]
//             modules: Module 1 (FSOES), Module 2 (DO)
//           Klemme 12 (EL7332) [EL7332 2K. DC-Motor-Endstufe (24V, 1.5A)]
//           Klemme 13 (EL3062-0030) [EL3062-0030 2K.Ana. Eingang 0-30V]
//           Klemme 14 (EL1004) [EL1004 4K. Dig. Eingang 24V, 3ms]
//           Klemme 15 (EL2004) [EL2004 4K. Dig. Ausgang 24V, 0.5A]
//           Klemme 51 (EL1104)
//           Klemme 16 (EL9010) [EL9010 Endklemme]
//         Oven_B (EK1100) [EK1100 EtherCAT-Koppler (2A E-Bus)]
//           Klemme 18 (EL1904) [EL1904, 4 K. Safety Eingang 24V, TwinSAFE]
//             modules: Module 1 (FSOES)
//           Klemme 19 (EL2904) [EL2904, 4 K. Safety Ausgang 24V, 0.5A, TwinSAFE]
//             modules: Module 1 (FSOES), Module 2 (DO)
//           Klemme 20 (EL7332) [EL7332 2K. DC-Motor-Endstufe (24V, 1.5A)]
//           Klemme 21 (EL3062-0030) [EL3062-0030 2K.Ana. Eingang 0-30V]
//           Klemme 22 (EL1004) [EL1004 4K. Dig. Eingang 24V, 3ms]
//           Klemme 23 (EL2004) [EL2004 4K. Dig. Ausgang 24V, 0.5A]
//           Klemme 66 (EL1104)
//           Klemme 61 (EL9010) [EL9010 Endklemme]
//       Storage|Casting (EK1122) [EK1122 2-Port EtherCAT-Abzweig]
//         Box 24 (EL6695-0002) [EL6695 EtherCAT Bridge terminal (Secondary)]
//         Storage (EK1100)
//       Klemme 83 (EL9410)
//       Term 71 (EL1008) [EL1008 8Ch. Dig. Input 24V, 3ms]
//       Term 73 (EL1008) [EL1008 8Ch. Dig. Input 24V, 3ms]
//       Term 74 (EL2008) [EL2008 8K. Dig. Ausgang 24V, 0.5A]
//       Term 75 (EL2008) [EL2008 8Ch. Dig. Output 24V, 0.5A]
//       Term 76 (EL1904) [EL1904, 4 Ch. Safety Input 24V, TwinSAFE]
//         modules: Module 1 (FSOES)
//       Klemme 93 (EL6070-0033)
//       Term 84 (EL9011) [EL9011 End Terminal]
//     RackFeeder_X_Y (AX5206-0000-0215) [AX5206-0000-0215 EtherCAT Drive (SoE, 2 Ch.)]
//       Klemme 27 (AX5805) [AX5805 (Safety Drive Option)]
//         modules: Module 1 (Safety Process Data, 2 axis), Module 2 (Standard Process Data, 2 axis)
//     Rackfeeder_Teleskop (AX5203-0000-0215) [AX5203-0000-0215 EtherCAT Drive (SoE, 2 Ch.)]
//       Klemme 29 (AX5805) [AX5805 (Safety Drive Option)]
//         modules: Module 1 (Safety Process Data, 2 axis), Module 2 (Standard Process Data, 2 axis)
//     OvenDoor_A_B (AX5206-0000-0215) [AX5206-0000-0215 EtherCAT Drive (SoE, 2 Ch.)]
//       Klemme 31 (AX5805) [AX5805 (Safety Drive Option)]
//         modules: Module 1 (Safety Process Data, 2 axis), Module 2 (Standard Process Data, 2 axis)
// variable links:
//   Device 3 (EtherCAT) <-> Device 3 (EtherCAT)/OvenDoor_A_B (AX5206-0000-0215)/Term 31 (AX5805)
//     Term 1 (EK1100)/Term 33 (EL6910)/ConnectionInputs/TwinSafeMain.Oven (AX5805) - Module 1 (Safety Process Data, 2 axis)_120 TxPDO <-> Module 1 (Safety Process Data, 2 axis)/Outputs (Controlword)/FSOE
//     Term 1 (EK1100)/Term 33 (EL6910)/ConnectionOutputs/TwinSafeMain.Oven (AX5805) - Module 1 (Safety Process Data, 2 axis)_120 RxPDO <-> Module 1 (Safety Process Data, 2 axis)/Inputs (Statusword)/FSOE
//   Device 3 (EtherCAT) <-> Device 3 (EtherCAT)/RackFeeder_X_Y (AX5206-0000-0215)/Term 27 (AX5805)
//     Term 1 (EK1100)/Term 33 (EL6910)/ConnectionInputs/TwinSafeMain.Rackfeeder_XY (AX5805) - Module 1 (Safety Process Data, 2 axis)_118 TxPDO <-> Module 1 (Safety Process Data, 2 axis)/Outputs (Controlword)/FSOE
//     Term 1 (EK1100)/Term 33 (EL6910)/ConnectionOutputs/TwinSafeMain.Rackfeeder_XY (AX5805) - Module 1 (Safety Process Data, 2 axis)_118 RxPDO <-> Module 1 (Safety Process Data, 2 axis)/Inputs (Statusword)/FSOE
//   Device 3 (EtherCAT) <-> Device 3 (EtherCAT)/Rackfeeder_Teleskop (AX5203-0000-0215)/Term 29 (AX5805)
//     Term 1 (EK1100)/Term 33 (EL6910)/ConnectionInputs/TwinSafeMain.Rackfeeder_Tele (AX5805) - Module 1 (Safety Process Data, 2 axis)_119 TxPDO <-> Module 1 (Safety Process Data, 2 axis)/Outputs (Controlword)/FSOE
//   Device 3 (EtherCAT) <-> Device 3 (EtherCAT)/Term 1 (EK1100)/Ovens (EK1122)/Oven_A (EK1100)/Term 10 (EL1904)
//     Term 1 (EK1100)/Term 33 (EL6910)/ConnectionInputs/TwinSafeMain.Oven A (EL1904) - Module 1 (FSOES)_14 TxPDO <-> Module 1 (FSOES)/RxPDO/FSOE
//     Term 1 (EK1100)/Term 33 (EL6910)/ConnectionOutputs/TwinSafeMain.Oven A (EL1904) - Module 1 (FSOES)_14 RxPDO <-> Module 1 (FSOES)/TxPDO/FSOE
//   Device 3 (EtherCAT) <-> Device 3 (EtherCAT)/Term 1 (EK1100)/Ovens (EK1122)/Oven_A (EK1100)/Term 11 (EL2904)
//     Term 1 (EK1100)/Term 33 (EL6910)/ConnectionInputs/TwinSafeMain.Oven A (EL2904) - Module 1 (FSOES)_111 TxPDO <-> Module 1 (FSOES)/RxPDO/FSOE
//     Term 1 (EK1100)/Term 33 (EL6910)/ConnectionOutputs/TwinSafeMain.Oven A (EL2904) - Module 1 (FSOES)_111 RxPDO <-> Module 1 (FSOES)/TxPDO/FSOE
//   Device 3 (EtherCAT) <-> Device 3 (EtherCAT)/Term 1 (EK1100)/Ovens (EK1122)/Oven_B (EK1100)/Term 18 (EL1904)
//     Term 1 (EK1100)/Term 33 (EL6910)/ConnectionInputs/TwinSafeMain.Oven B (EL1904) - Module 1 (FSOES)_16 TxPDO <-> Module 1 (FSOES)/RxPDO/FSOE
//     Term 1 (EK1100)/Term 33 (EL6910)/ConnectionOutputs/TwinSafeMain.Oven B (EL1904) - Module 1 (FSOES)_16 RxPDO <-> Module 1 (FSOES)/TxPDO/FSOE
//   Device 3 (EtherCAT) <-> Device 3 (EtherCAT)/Term 1 (EK1100)/Ovens (EK1122)/Oven_B (EK1100)/Term 19 (EL2904)
//     Term 1 (EK1100)/Term 33 (EL6910)/ConnectionInputs/TwinSafeMain.Oven B (EL2904) - Module 1 (FSOES)_112 TxPDO <-> Module 1 (FSOES)/RxPDO/FSOE
//     Term 1 (EK1100)/Term 33 (EL6910)/ConnectionOutputs/TwinSafeMain.Oven B (EL2904) - Module 1 (FSOES)_112 RxPDO <-> Module 1 (FSOES)/TxPDO/FSOE
//   Device 3 (EtherCAT) <-> Device 3 (EtherCAT)/Term 1 (EK1100)/Term 3 (EL1904)
//     Term 1 (EK1100)/Term 33 (EL6910)/ConnectionInputs/TwinSafeMain.MAIN (EL1904) - Module 1 (FSOES)_12 TxPDO <-> Module 1 (FSOES)/RxPDO/FSOE
//     Term 1 (EK1100)/Term 33 (EL6910)/ConnectionOutputs/TwinSafeMain.MAIN (EL1904) - Module 1 (FSOES)_12 RxPDO <-> Module 1 (FSOES)/TxPDO/FSOE
//   Device 3 (EtherCAT) <-> Device 3 (EtherCAT)/Term 1 (EK1100)/Term 33 (EL6910)
//     Rackfeeder_Teleskop (AX5203-0000-0215)/Term 29 (AX5805)/Module 1 (Safety Process Data, 2 axis)/Inputs (Statusword)/FSOE <-> ConnectionOutputs/TwinSafeMain.Rackfeeder_Tele (AX5805) - Module 1 (Safety Process Data, 2 axis)_119 RxPDO
//     Term 1 (EK1100)/Term 43 (EL1904)/Module 1 (FSOES)/RxPDO/FSOE <-> ConnectionInputs/TwinSafeMain.MAIN (EL1904_2) - Module 1 (FSOES)_135 TxPDO
//     Term 1 (EK1100)/Term 76 (EL1904)/Module 1 (FSOES)/TxPDO/FSOE <-> ConnectionOutputs/TwinSafeMain.EUCHNER (EL1904) - Module 1 (FSOES)_136 RxPDO
//   Device 3 (EtherCAT) <-> Device 3 (EtherCAT)/Term 1 (EK1100)/Term 4 (EL2904)
//     Term 1 (EK1100)/Term 33 (EL6910)/ConnectionInputs/TwinSafeMain.MAIN (EL2904) - Module 1 (FSOES)_13 TxPDO <-> Module 1 (FSOES)/RxPDO/FSOE
//     Term 1 (EK1100)/Term 33 (EL6910)/ConnectionOutputs/TwinSafeMain.MAIN (EL2904) - Module 1 (FSOES)_13 RxPDO <-> Module 1 (FSOES)/TxPDO/FSOE
//   Device 3 (EtherCAT) <-> Device 3 (EtherCAT)/Term 1 (EK1100)/Term 43 (EL1904)
//     Term 1 (EK1100)/Term 33 (EL6910)/ConnectionOutputs/TwinSafeMain.MAIN (EL1904_2) - Module 1 (FSOES)_135 RxPDO <-> Module 1 (FSOES)/TxPDO/FSOE
//   Device 3 (EtherCAT) <-> Device 3 (EtherCAT)/Term 1 (EK1100)/Term 76 (EL1904)
//     Term 1 (EK1100)/Term 33 (EL6910)/ConnectionInputs/TwinSafeMain.EUCHNER (EL1904) - Module 1 (FSOES)_136 TxPDO <-> Module 1 (FSOES)/RxPDO/FSOE
//   NC-Task 1 SAF/Axes/Oven A <-> Device 3 (EtherCAT)/OvenDoor_A_B (AX5206-0000-0215)
//     Drive/Inputs/In/nDataIn1 <-> AT 1/Following distance
//     Drive/Inputs/In/nDataIn3[0] <-> AT 1/Torque/force feedback value
//     Drive/Inputs/In/nDcOutputTime <-> InfoData/DcOutputShift
//     Drive/Inputs/In/nState1 <-> AT 1/Drive status word @bit 8
//     Drive/Inputs/In/nState2 <-> AT 1/Drive status word
//     Drive/Inputs/In/nState4 @bit 1 <-> WcState/InputToggle
//     Drive/Inputs/In/nState4 <-> WcState/WcState
//     Drive/Outputs/Out/nCtrl1 <-> MDT 1/Master control word @bit 8
//     Drive/Outputs/Out/nDataOut1 <-> MDT 1/Position command value
//     Enc/Inputs/In/nDataIn1 <-> AT 1/Position feedback 1 value
//     Enc/Inputs/In/nDcInputTime <-> InfoData/DcInputShift
//     Enc/Inputs/In/nState4 @bit 1 <-> WcState/InputToggle
//     Enc/Inputs/In/nState4 <-> WcState/WcState
//   NC-Task 1 SAF/Axes/Oven A CH1 <-> Device 3 (EtherCAT)/Term 1 (EK1100)/Ovens (EK1122)/Oven_A (EK1100)/Term 12 (EL7332)
//     Drive/Inputs/In/nState1 @bit 3 <-> DCM Status Channel 1/Status/Error
//     Drive/Inputs/In/nState1 @bit 5 <-> DCM Status Channel 1/Status/Moving negative
//     Drive/Inputs/In/nState1 @bit 4 <-> DCM Status Channel 1/Status/Moving positive
//     Drive/Inputs/In/nState1 @bit 1 <-> DCM Status Channel 1/Status/Ready
//     Drive/Inputs/In/nState1 <-> DCM Status Channel 1/Status/Ready to enable
//     Drive/Inputs/In/nState1 @bit 6 <-> DCM Status Channel 1/Status/Torque reduced
//     Drive/Inputs/In/nState1 @bit 2 <-> DCM Status Channel 1/Status/Warning
//     Drive/Inputs/In/nState2 @bit 3 <-> DCM Status Channel 1/Status/Digital input 1
//     Drive/Inputs/In/nState2 @bit 4 <-> DCM Status Channel 1/Status/Digital input 2
//     Drive/Inputs/In/nState2 @bit 5 <-> DCM Status Channel 1/Status/Sync error
//     Drive/Inputs/In/nState2 @bit 7 <-> DCM Status Channel 1/Status/TxPDO Toggle
//     Drive/Inputs/In/nState4 @bit 1 <-> WcState/InputToggle
//     Drive/Inputs/In/nState4 <-> WcState/WcState
//     Drive/Outputs/Out/nCtrl1 <-> DCM Control Channel 1/Control/Enable
//     Drive/Outputs/Out/nCtrl1 @bit 2 <-> DCM Control Channel 1/Control/Reduce torque
//     Drive/Outputs/Out/nCtrl1 @bit 1 <-> DCM Control Channel 1/Control/Reset
//     Drive/Outputs/Out/nDataOut2[0] <-> DCM Velocity Channel 1/Velocity
//   NC-Task 1 SAF/Axes/Oven A CH1 <-> Device 3 (EtherCAT)/Term 1 (EK1100)/Ovens (EK1122)/Oven_A (EK1100)/Term 13 (EL3062-0030)
//     Enc/Inputs/In/nDataIn1[0] <-> AI Standard Channel 1/Value
//     Enc/Inputs/In/nState4 @bit 1 <-> WcState/InputToggle
//     Enc/Inputs/In/nState4 <-> WcState/WcState
//   NC-Task 1 SAF/Axes/Oven A CH2 <-> Device 3 (EtherCAT)/Term 1 (EK1100)/Ovens (EK1122)/Oven_A (EK1100)/Term 12 (EL7332)
//     Drive/Inputs/In/nState1 @bit 3 <-> DCM Status Channel 2/Status/Error
//     Drive/Inputs/In/nState1 @bit 5 <-> DCM Status Channel 2/Status/Moving negative
//     Drive/Inputs/In/nState1 @bit 4 <-> DCM Status Channel 2/Status/Moving positive
//     Drive/Inputs/In/nState1 @bit 1 <-> DCM Status Channel 2/Status/Ready
//     Drive/Inputs/In/nState1 <-> DCM Status Channel 2/Status/Ready to enable
//     Drive/Inputs/In/nState1 @bit 6 <-> DCM Status Channel 2/Status/Torque reduced
//     Drive/Inputs/In/nState1 @bit 2 <-> DCM Status Channel 2/Status/Warning
//     Drive/Inputs/In/nState2 @bit 3 <-> DCM Status Channel 2/Status/Digital input 1
//     Drive/Inputs/In/nState2 @bit 4 <-> DCM Status Channel 2/Status/Digital input 2
//     Drive/Inputs/In/nState2 @bit 5 <-> DCM Status Channel 2/Status/Sync error
//     Drive/Inputs/In/nState2 @bit 7 <-> DCM Status Channel 2/Status/TxPDO Toggle
//     Drive/Inputs/In/nState4 @bit 1 <-> WcState/InputToggle
//     Drive/Inputs/In/nState4 <-> WcState/WcState
//     Drive/Outputs/Out/nCtrl1 <-> DCM Control Channel 2/Control/Enable
//     Drive/Outputs/Out/nCtrl1 @bit 2 <-> DCM Control Channel 2/Control/Reduce torque
//     Drive/Outputs/Out/nCtrl1 @bit 1 <-> DCM Control Channel 2/Control/Reset
//     Drive/Outputs/Out/nDataOut2[0] <-> DCM Velocity Channel 2/Velocity
//   NC-Task 1 SAF/Axes/Oven A CH2 <-> Device 3 (EtherCAT)/Term 1 (EK1100)/Ovens (EK1122)/Oven_A (EK1100)/Term 13 (EL3062-0030)
//     Enc/Inputs/In/nDataIn1[0] <-> AI Standard Channel 2/Value
//     Enc/Inputs/In/nState4 @bit 1 <-> WcState/InputToggle
//     Enc/Inputs/In/nState4 <-> WcState/WcState
//   NC-Task 1 SAF/Axes/Oven B <-> Device 3 (EtherCAT)/OvenDoor_A_B (AX5206-0000-0215)
//     Drive/Inputs/In/nDataIn1 <-> AT 2/Following distance
//     Drive/Inputs/In/nDataIn3[0] <-> AT 2/Torque/force feedback value
//     Drive/Inputs/In/nDcOutputTime <-> InfoData/DcOutputShift
//     Drive/Inputs/In/nState1 <-> AT 2/Drive status word @bit 8
//     Drive/Inputs/In/nState2 <-> AT 2/Drive status word
//     Drive/Inputs/In/nState4 @bit 1 <-> WcState/InputToggle
//     Drive/Inputs/In/nState4 <-> WcState/WcState
//     Drive/Outputs/Out/nCtrl1 <-> MDT 2/Master control word @bit 8
//     Drive/Outputs/Out/nDataOut1 <-> MDT 2/Position command value
//     Enc/Inputs/In/nDataIn1 <-> AT 2/Position feedback 1 value
//     Enc/Inputs/In/nDcInputTime <-> InfoData/DcInputShift
//     Enc/Inputs/In/nState4 @bit 1 <-> WcState/InputToggle
//     Enc/Inputs/In/nState4 <-> WcState/WcState
//   NC-Task 1 SAF/Axes/Oven B CH1 <-> Device 3 (EtherCAT)/Term 1 (EK1100)/Ovens (EK1122)/Oven_B (EK1100)/Term 20 (EL7332)
//     Drive/Inputs/In/nState1 @bit 3 <-> DCM Status Channel 1/Status/Error
//     Drive/Inputs/In/nState1 @bit 5 <-> DCM Status Channel 1/Status/Moving negative
//     Drive/Inputs/In/nState1 @bit 4 <-> DCM Status Channel 1/Status/Moving positive
//     Drive/Inputs/In/nState1 @bit 1 <-> DCM Status Channel 1/Status/Ready
//     Drive/Inputs/In/nState1 <-> DCM Status Channel 1/Status/Ready to enable
//     Drive/Inputs/In/nState1 @bit 6 <-> DCM Status Channel 1/Status/Torque reduced
//     Drive/Inputs/In/nState1 @bit 2 <-> DCM Status Channel 1/Status/Warning
//     Drive/Inputs/In/nState2 @bit 3 <-> DCM Status Channel 1/Status/Digital input 1
//     Drive/Inputs/In/nState2 @bit 4 <-> DCM Status Channel 1/Status/Digital input 2
//     Drive/Inputs/In/nState2 @bit 5 <-> DCM Status Channel 1/Status/Sync error
//     Drive/Inputs/In/nState2 @bit 7 <-> DCM Status Channel 1/Status/TxPDO Toggle
//     Drive/Inputs/In/nState4 @bit 1 <-> WcState/InputToggle
//     Drive/Inputs/In/nState4 <-> WcState/WcState
//     Drive/Outputs/Out/nCtrl1 <-> DCM Control Channel 1/Control/Enable
//     Drive/Outputs/Out/nCtrl1 @bit 2 <-> DCM Control Channel 1/Control/Reduce torque
//     Drive/Outputs/Out/nCtrl1 @bit 1 <-> DCM Control Channel 1/Control/Reset
//     Drive/Outputs/Out/nDataOut2[0] <-> DCM Velocity Channel 1/Velocity
//   NC-Task 1 SAF/Axes/Oven B CH1 <-> Device 3 (EtherCAT)/Term 1 (EK1100)/Ovens (EK1122)/Oven_B (EK1100)/Term 21 (EL3062-0030)
//     Enc/Inputs/In/nDataIn1[0] <-> AI Standard Channel 1/Value
//     Enc/Inputs/In/nState4 @bit 1 <-> WcState/InputToggle
//     Enc/Inputs/In/nState4 <-> WcState/WcState
//   NC-Task 1 SAF/Axes/Oven B CH2 <-> Device 3 (EtherCAT)/Term 1 (EK1100)/Ovens (EK1122)/Oven_B (EK1100)/Term 20 (EL7332)
//     Drive/Inputs/In/nState1 @bit 3 <-> DCM Status Channel 2/Status/Error
//     Drive/Inputs/In/nState1 @bit 5 <-> DCM Status Channel 2/Status/Moving negative
//     Drive/Inputs/In/nState1 @bit 4 <-> DCM Status Channel 2/Status/Moving positive
//     Drive/Inputs/In/nState1 @bit 1 <-> DCM Status Channel 2/Status/Ready
//     Drive/Inputs/In/nState1 <-> DCM Status Channel 2/Status/Ready to enable
//     Drive/Inputs/In/nState1 @bit 6 <-> DCM Status Channel 2/Status/Torque reduced
//     Drive/Inputs/In/nState1 @bit 2 <-> DCM Status Channel 2/Status/Warning
//     Drive/Inputs/In/nState2 @bit 3 <-> DCM Status Channel 2/Status/Digital input 1
//     Drive/Inputs/In/nState2 @bit 4 <-> DCM Status Channel 2/Status/Digital input 2
//     Drive/Inputs/In/nState2 @bit 5 <-> DCM Status Channel 2/Status/Sync error
//     Drive/Inputs/In/nState2 @bit 7 <-> DCM Status Channel 2/Status/TxPDO Toggle
//     Drive/Inputs/In/nState4 @bit 1 <-> WcState/InputToggle
//     Drive/Inputs/In/nState4 <-> WcState/WcState
//     Drive/Outputs/Out/nCtrl1 <-> DCM Control Channel 2/Control/Enable
//     Drive/Outputs/Out/nCtrl1 @bit 2 <-> DCM Control Channel 2/Control/Reduce torque
//     Drive/Outputs/Out/nCtrl1 @bit 1 <-> DCM Control Channel 2/Control/Reset
//     Drive/Outputs/Out/nDataOut2[0] <-> DCM Velocity Channel 2/Velocity
//   NC-Task 1 SAF/Axes/Oven B CH2 <-> Device 3 (EtherCAT)/Term 1 (EK1100)/Ovens (EK1122)/Oven_B (EK1100)/Term 21 (EL3062-0030)
//     Enc/Inputs/In/nDataIn1[0] <-> AI Standard Channel 2/Value
//     Enc/Inputs/In/nState4 @bit 1 <-> WcState/InputToggle
//     Enc/Inputs/In/nState4 <-> WcState/WcState
//   NC-Task 1 SAF/Axes/Rackfeeder X <-> Device 3 (EtherCAT)/RackFeeder_X_Y (AX5206-0000-0215)
//     Drive/Inputs/In/nDataIn1 <-> AT 1/Following distance
//     Drive/Inputs/In/nDataIn3[0] <-> AT 1/Torque/force feedback value
//     Drive/Inputs/In/nDcOutputTime <-> InfoData/DcOutputShift
//     Drive/Inputs/In/nState1 <-> AT 1/Drive status word @bit 8
//     Drive/Inputs/In/nState2 <-> AT 1/Drive status word
//     Drive/Inputs/In/nState4 @bit 1 <-> WcState/InputToggle
//     Drive/Inputs/In/nState4 <-> WcState/WcState
//     Drive/Outputs/Out/nCtrl1 <-> MDT 1/Master control word @bit 8
//     Drive/Outputs/Out/nDataOut1 <-> MDT 1/Position command value
//     Enc/Inputs/In/nDataIn1 <-> AT 1/Position feedback 1 value
//     Enc/Inputs/In/nDcInputTime <-> InfoData/DcInputShift
//     Enc/Inputs/In/nState4 @bit 1 <-> WcState/InputToggle
//     Enc/Inputs/In/nState4 <-> WcState/WcState
//   NC-Task 1 SAF/Axes/Rackfeeder Y <-> Device 3 (EtherCAT)/RackFeeder_X_Y (AX5206-0000-0215)
//     Drive/Inputs/In/nDataIn1 <-> AT 2/Following distance
//     Drive/Inputs/In/nDataIn3[0] <-> AT 2/Torque/force feedback value
//     Drive/Inputs/In/nDcOutputTime <-> InfoData/DcOutputShift
//     Drive/Inputs/In/nState1 <-> AT 2/Drive status word @bit 8
//     Drive/Inputs/In/nState2 <-> AT 2/Drive status word
//     Drive/Inputs/In/nState4 @bit 1 <-> WcState/InputToggle
//     Drive/Inputs/In/nState4 <-> WcState/WcState
//     Drive/Outputs/Out/nCtrl1 <-> MDT 2/Master control word @bit 8
//     Drive/Outputs/Out/nDataOut1 <-> MDT 2/Position command value
//     Enc/Inputs/In/nDataIn1 <-> AT 2/Position feedback 1 value
//     Enc/Inputs/In/nDcInputTime <-> InfoData/DcInputShift
//     Enc/Inputs/In/nState4 @bit 1 <-> WcState/InputToggle
//     Enc/Inputs/In/nState4 <-> WcState/WcState
//   NC-Task 1 SAF/Axes/Rackfeeder Z <-> Device 3 (EtherCAT)/Rackfeeder_Teleskop (AX5203-0000-0215)
//     Drive/Inputs/In/nDataIn1 <-> AT 1/Following distance
//     Drive/Inputs/In/nDataIn3[0] <-> AT 1/Torque/force feedback value
//     Drive/Inputs/In/nDcOutputTime <-> InfoData/DcOutputShift
//     Drive/Inputs/In/nState1 <-> AT 1/Drive status word @bit 8
//     Drive/Inputs/In/nState2 <-> AT 1/Drive status word
//     Drive/Inputs/In/nState4 @bit 1 <-> WcState/InputToggle
//     Drive/Inputs/In/nState4 <-> WcState/WcState
//     Drive/Outputs/Out/nCtrl1 <-> MDT 1/Master control word @bit 8
//     Drive/Outputs/Out/nDataOut1 <-> MDT 1/Position command value
//     Enc/Inputs/In/nDataIn1 <-> AT 1/Position feedback 1 value
//     Enc/Inputs/In/nDcInputTime <-> InfoData/DcInputShift
//     Enc/Inputs/In/nState4 @bit 1 <-> WcState/InputToggle
//     Enc/Inputs/In/nState4 <-> WcState/WcState
//   NC-Task 1 SAF/Axes/Storage A <-> Device 3 (EtherCAT)/Term 1 (EK1100)/Storage|Casting (EK1122)/Storage (EK1100)/Term 63 (EL3062)
//     Enc/Inputs/In/nDataIn1[0] <-> AI Standard Channel 1/Value
//     Enc/Inputs/In/nState4 @bit 1 <-> WcState/InputToggle
//     Enc/Inputs/In/nState4 <-> WcState/WcState
//   NC-Task 1 SAF/Axes/Storage A <-> Device 3 (EtherCAT)/Term 1 (EK1100)/Storage|Casting (EK1122)/Storage (EK1100)/Term 64 (EL7332)
//     Drive/Inputs/In/nState1 @bit 3 <-> DCM Status Channel 1/Status/Error
//     Drive/Inputs/In/nState1 @bit 5 <-> DCM Status Channel 1/Status/Moving negative
//     Drive/Inputs/In/nState1 @bit 4 <-> DCM Status Channel 1/Status/Moving positive
//     Drive/Inputs/In/nState1 @bit 1 <-> DCM Status Channel 1/Status/Ready
//     Drive/Inputs/In/nState1 <-> DCM Status Channel 1/Status/Ready to enable
//     Drive/Inputs/In/nState1 @bit 6 <-> DCM Status Channel 1/Status/Torque reduced
//     Drive/Inputs/In/nState1 @bit 2 <-> DCM Status Channel 1/Status/Warning
//     Drive/Inputs/In/nState2 @bit 3 <-> DCM Status Channel 1/Status/Digital input 1
//     Drive/Inputs/In/nState2 @bit 4 <-> DCM Status Channel 1/Status/Digital input 2
//     Drive/Inputs/In/nState2 @bit 5 <-> DCM Status Channel 1/Status/Sync error
//     Drive/Inputs/In/nState2 @bit 7 <-> DCM Status Channel 1/Status/TxPDO Toggle
//     Drive/Inputs/In/nState4 @bit 1 <-> WcState/InputToggle
//     Drive/Inputs/In/nState4 <-> WcState/WcState
//     Drive/Outputs/Out/nCtrl1 <-> DCM Control Channel 1/Control/Enable
//     Drive/Outputs/Out/nCtrl1 @bit 2 <-> DCM Control Channel 1/Control/Reduce torque
//     Drive/Outputs/Out/nCtrl1 @bit 1 <-> DCM Control Channel 1/Control/Reset
//     Drive/Outputs/Out/nDataOut2[0] <-> DCM Velocity Channel 1/Velocity
//   NC-Task 1 SAF/Axes/Storage B <-> Device 3 (EtherCAT)/Term 1 (EK1100)/Storage|Casting (EK1122)/Storage (EK1100)/Term 63 (EL3062)
//     Enc/Inputs/In/nDataIn1[0] <-> AI Standard Channel 2/Value
//     Enc/Inputs/In/nState4 @bit 1 <-> WcState/InputToggle
//     Enc/Inputs/In/nState4 <-> WcState/WcState
//   NC-Task 1 SAF/Axes/Storage B <-> Device 3 (EtherCAT)/Term 1 (EK1100)/Storage|Casting (EK1122)/Storage (EK1100)/Term 64 (EL7332)
//     Drive/Inputs/In/nState1 @bit 3 <-> DCM Status Channel 2/Status/Error
//     Drive/Inputs/In/nState1 @bit 5 <-> DCM Status Channel 2/Status/Moving negative
//     Drive/Inputs/In/nState1 @bit 4 <-> DCM Status Channel 2/Status/Moving positive
//     Drive/Inputs/In/nState1 @bit 1 <-> DCM Status Channel 2/Status/Ready
//     Drive/Inputs/In/nState1 <-> DCM Status Channel 2/Status/Ready to enable
//     Drive/Inputs/In/nState1 @bit 6 <-> DCM Status Channel 2/Status/Torque reduced
//     Drive/Inputs/In/nState1 @bit 2 <-> DCM Status Channel 2/Status/Warning
//     Drive/Inputs/In/nState2 @bit 3 <-> DCM Status Channel 2/Status/Digital input 1
//     Drive/Inputs/In/nState2 @bit 4 <-> DCM Status Channel 2/Status/Digital input 2
//     Drive/Inputs/In/nState2 @bit 5 <-> DCM Status Channel 2/Status/Sync error
//     Drive/Inputs/In/nState2 @bit 7 <-> DCM Status Channel 2/Status/TxPDO Toggle
//     Drive/Inputs/In/nState4 @bit 1 <-> WcState/InputToggle
//     Drive/Inputs/In/nState4 <-> WcState/WcState
//     Drive/Outputs/Out/nCtrl1 <-> DCM Control Channel 2/Control/Enable
//     Drive/Outputs/Out/nCtrl1 @bit 2 <-> DCM Control Channel 2/Control/Reduce torque
//     Drive/Outputs/Out/nCtrl1 @bit 1 <-> DCM Control Channel 2/Control/Reset
//     Drive/Outputs/Out/nDataOut2[0] <-> DCM Velocity Channel 2/Velocity
//   PLC/PLC Instance <-> Device 3 (EtherCAT)
//     PlcTask Inputs/IO.stControlCabinetIO.stIn/eEtherCATDeviceState <-> Inputs/DevState
//     PlcTask Inputs/IO.stControlCabinetIO.stIn/stEtherCATMasterAmsAdr/netId <-> InfoData/AmsNetId
//     PlcTask Inputs/IO.stControlCabinetIO.stIn/uiEcMasterDevId <-> InfoData/DevId
//     PlcTask Inputs/P_Supervision.fbDiagEtherCAT.aEcMasters[0]/nDevId <-> InfoData/DevId
//     PlcTask Inputs/P_Supervision.fbDiagEtherCAT.aEcMasters[0]/nDeviceState <-> Inputs/DevState
//     PlcTask Inputs/P_Supervision.fbDiagEtherCAT.aEcMasters[0]/stAmsAdr/netId <-> InfoData/AmsNetId
//   PLC/PLC Instance <-> Device 3 (EtherCAT)/OvenDoor_A_B (AX5206-0000-0215)
//     PlcTask Outputs/NcIO.stAxis_ST010_OvenA_IO.stOut/iBipolarTorqueLimitValue <-> MDT 1/Bipolar torque/force limit value
//     PlcTask Outputs/NcIO.stAxis_ST020_OvenB_IO.stOut/iBipolarTorqueLimitValue <-> MDT 2/Bipolar torque/force limit value
//   PLC/PLC Instance <-> Device 3 (EtherCAT)/RackFeeder_X_Y (AX5206-0000-0215)
//     PlcTask Outputs/NcIO.stAxis_ST030_AxisX_IO.stOut/iBipolarTorqueLimitValue <-> MDT 1/Bipolar torque/force limit value
//     PlcTask Outputs/NcIO.stAxis_ST030_AxisY_IO.stOut/iBipolarTorqueLimitValue <-> MDT 2/Bipolar torque/force limit value
//   PLC/PLC Instance <-> Device 3 (EtherCAT)/Rackfeeder_Teleskop (AX5203-0000-0215)
//     PlcTask Outputs/NcIO.stAxis_ST030_AxisZ_IO.stOut/iBipolarTorqueLimitValue <-> MDT 1/Bipolar torque/force limit value
//   PLC/PLC Instance <-> Device 3 (EtherCAT)/Term 1 (EK1100)
//     PlcTask Inputs/IO.stControlCabinetIO.stIn/IarrEcStates[0] <-> InfoData/State
//   PLC/PLC Instance <-> Device 3 (EtherCAT)/Term 1 (EK1100)/Ovens (EK1122)/Oven_A (EK1100)
//     PlcTask Inputs/IO.stControlCabinetIO.stIn/IarrEcStates[1] <-> InfoData/State
//   PLC/PLC Instance <-> Device 3 (EtherCAT)/Term 1 (EK1100)/Ovens (EK1122)/Oven_A (EK1100)/Term 14 (EL1004)
//     PlcTask Inputs/IO.st010_OvenA_IO.stIn/bRefpos <-> Channel 4/bRefpos
//     PlcTask Inputs/Safety.arrSaftyDoors[0].stHwIn/bLockButton <-> Channel 3/bLockButton
//     PlcTask Inputs/Safety.arrSaftyDoors[0].stHwIn/bRequestButton <-> Channel 2/bRequestButton
//     PlcTask Inputs/Safety.arrSaftyDoors[0].stHwIn/bStartButton <-> Channel 1/bStartButton
//   PLC/PLC Instance <-> Device 3 (EtherCAT)/Term 1 (EK1100)/Ovens (EK1122)/Oven_A (EK1100)/Term 15 (EL2004)
//     PlcTask Outputs/Safety.arrSaftyDoors[0].stHwOut/bLockLight <-> Channel 3/bLockLight
//     PlcTask Outputs/Safety.arrSaftyDoors[0].stHwOut/bStartLight <-> Channel 1/bStartLight
//     PlcTask Outputs/Safety.arrSaftyDoors[0].stHwOut/bStopLight <-> Channel 2/bRequestLight
//   PLC/PLC Instance <-> Device 3 (EtherCAT)/Term 1 (EK1100)/Ovens (EK1122)/Oven_A (EK1100)/Term 51 (EL1104)
//     PlcTask Inputs/Safety.arrSaftyDoors[0].stHwIn/bLocked <-> Channel 1/Input
//   PLC/PLC Instance <-> Device 3 (EtherCAT)/Term 1 (EK1100)/Ovens (EK1122)/Oven_B (EK1100)
//     PlcTask Inputs/IO.stControlCabinetIO.stIn/IarrEcStates[2] <-> InfoData/State
//   PLC/PLC Instance <-> Device 3 (EtherCAT)/Term 1 (EK1100)/Ovens (EK1122)/Oven_B (EK1100)/Term 22 (EL1004)
//     PlcTask Inputs/IO.st020_OvenB_IO.stIn/bRefpos <-> Channel 4/bRefpos
//     PlcTask Inputs/Safety.arrSaftyDoors[1].stHwIn/bLockButton <-> Channel 3/bLockButton
//     PlcTask Inputs/Safety.arrSaftyDoors[1].stHwIn/bRequestButton <-> Channel 2/bRequestButton
//     PlcTask Inputs/Safety.arrSaftyDoors[1].stHwIn/bStartButton <-> Channel 1/bStartButton
//   PLC/PLC Instance <-> Device 3 (EtherCAT)/Term 1 (EK1100)/Ovens (EK1122)/Oven_B (EK1100)/Term 23 (EL2004)
//     PlcTask Outputs/Safety.arrSaftyDoors[1].stHwOut/bLockLight <-> Channel 3/bLockLight
//     PlcTask Outputs/Safety.arrSaftyDoors[1].stHwOut/bStartLight <-> Channel 1/bStartLight
//     PlcTask Outputs/Safety.arrSaftyDoors[1].stHwOut/bStopLight <-> Channel 2/bRequestLight
//   PLC/PLC Instance <-> Device 3 (EtherCAT)/Term 1 (EK1100)/Ovens (EK1122)/Oven_B (EK1100)/Term 66 (EL1104)
//     PlcTask Inputs/Safety.arrSaftyDoors[1].stHwIn/bLocked <-> Channel 1/Input
//   PLC/PLC Instance <-> Device 3 (EtherCAT)/Term 1 (EK1100)/Storage|Casting (EK1122)/Box 24 (EL6695-0002)
//     PlcTask Inputs/IO.st050_Mould_IO.stIn/aFromEngelRaw <-> IO Inputs/Var 7820
//     PlcTask Inputs/IO.st050_Mould_IO.stIn/aFromEngelRaw @bit 16 <-> IO Inputs/Var 7821
//     PlcTask Inputs/IO.st050_Mould_IO.stIn/aFromEngelRaw @bit 32 <-> IO Inputs/Var 7822
//     PlcTask Inputs/IO.st050_Mould_IO.stIn/aFromEngelRaw @bit 33 <-> IO Inputs/Var 7823
//     PlcTask Inputs/IO.st050_Mould_IO.stIn/aFromEngelRaw @bit 34 <-> IO Inputs/Var 7824
//     PlcTask Inputs/IO.st050_Mould_IO.stIn/aFromEngelRaw @bit 35 <-> IO Inputs/Var 7825
//     PlcTask Inputs/IO.st050_Mould_IO.stIn/aFromEngelRaw @bit 36 <-> IO Inputs/Var 7826
//     PlcTask Inputs/IO.st050_Mould_IO.stIn/aFromEngelRaw @bit 37 <-> IO Inputs/Var 7827
//     PlcTask Inputs/IO.st050_Mould_IO.stIn/aFromEngelRaw @bit 38 <-> IO Inputs/Var 7828
//     PlcTask Inputs/IO.st050_Mould_IO.stIn/aFromEngelRaw @bit 39 <-> IO Inputs/Var 7829
//     PlcTask Inputs/IO.st050_Mould_IO.stIn/aFromEngelRaw @bit 40 <-> IO Inputs/Var 7830
//     PlcTask Inputs/IO.st050_Mould_IO.stIn/aFromEngelRaw @bit 41 <-> IO Inputs/Var 7831
//     PlcTask Inputs/IO.st050_Mould_IO.stIn/aFromEngelRaw @bit 42 <-> IO Inputs/Var 7832
//     PlcTask Inputs/IO.st050_Mould_IO.stIn/aFromEngelRaw @bit 43 <-> IO Inputs/Var 7833
//     PlcTask Inputs/IO.st050_Mould_IO.stIn/aFromEngelRaw @bit 44 <-> IO Inputs/Var 7834
//     PlcTask Inputs/IO.st050_Mould_IO.stIn/aFromEngelRaw @bit 45 <-> IO Inputs/Var 7835
//     PlcTask Inputs/IO.st050_Mould_IO.stIn/aFromEngelRaw @bit 46 <-> IO Inputs/Var 7836
//     PlcTask Inputs/IO.st050_Mould_IO.stIn/aFromEngelRaw @bit 47 <-> IO Inputs/Var 7837
//     PlcTask Inputs/IO.st050_Mould_IO.stIn/aFromEngelRaw @bit 48 <-> IO Inputs/Var 7838
//     PlcTask Inputs/IO.st050_Mould_IO.stIn/aFromEngelRaw @bit 49 <-> IO Inputs/Var 7839
//     PlcTask Inputs/IO.st050_Mould_IO.stIn/aFromEngelRaw @bit 50 <-> IO Inputs/Var 7840
//     PlcTask Inputs/IO.st050_Mould_IO.stIn/aFromEngelRaw @bit 51 <-> IO Inputs/Var 7841
//     PlcTask Inputs/IO.st050_Mould_IO.stIn/aFromEngelRaw @bit 52 <-> IO Inputs/Var 7842
//     PlcTask Inputs/IO.st050_Mould_IO.stIn/aFromEngelRaw @bit 53 <-> IO Inputs/Var 7843
//     PlcTask Inputs/IO.st050_Mould_IO.stIn/aFromEngelRaw @bit 54 <-> IO Inputs/Var 7844
//     PlcTask Inputs/IO.st050_Mould_IO.stIn/aFromEngelRaw @bit 55 <-> IO Inputs/Var 7845
//     PlcTask Inputs/IO.st050_Mould_IO.stIn/aFromEngelRaw @bit 56 <-> IO Inputs/Var 7846
//     PlcTask Inputs/IO.st050_Mould_IO.stIn/aFromEngelRaw @bit 72 <-> IO Inputs/Var 7847
//     PlcTask Inputs/IO.st050_Mould_IO.stIn/aFromEngelRaw @bit 88 <-> IO Inputs/Var 7848
//     PlcTask Inputs/IO.st050_Mould_IO.stIn/aFromEngelRaw @bit 104 <-> IO Inputs/Var 7849
//     PlcTask Inputs/IO.st050_Mould_IO.stIn/aFromEngelRaw @bit 120 <-> IO Inputs/Var 7850
//     PlcTask Inputs/IO.st050_Mould_IO.stIn/aFromEngelRaw @bit 136 <-> IO Inputs/Var 7851
//     PlcTask Inputs/IO.st050_Mould_IO.stIn/aFromEngelRaw @bit 152 <-> IO Inputs/Var 7852
//     PlcTask Inputs/IO.st050_Mould_IO.stIn/aFromEngelRaw @bit 168 <-> IO Inputs/Var 7853
//     PlcTask Inputs/IO.st050_Mould_IO.stIn/aFromEngelRaw @bit 184 <-> IO Inputs/Var 7854
//     PlcTask Inputs/IO.st050_Mould_IO.stIn/aFromEngelRaw @bit 200 <-> IO Inputs/Var 7855
//     PlcTask Inputs/IO.st050_Mould_IO.stIn/aFromEngelRaw @bit 216 <-> IO Inputs/Var 7856
//     PlcTask Inputs/IO.st050_Mould_IO.stIn/aFromEngelRaw @bit 232 <-> IO Inputs/Var 7857
//     PlcTask Inputs/IO.st050_Mould_IO.stIn/aFromEngelRaw @bit 248 <-> IO Inputs/Var 7858
//     PlcTask Inputs/IO.st050_Mould_IO.stIn/aFromEngelRaw @bit 264 <-> IO Inputs/Var 7859
//     PlcTask Inputs/IO.st050_Mould_IO.stIn/aFromEngelRaw @bit 280 <-> IO Inputs/Var 7860
//     PlcTask Inputs/IO.st050_Mould_IO.stIn/aFromEngelRaw @bit 296 <-> IO Inputs/Var 7861
//     PlcTask Inputs/IO.st050_Mould_IO.stIn/aFromEngelRaw @bit 312 <-> IO Inputs/Var 7862
//     PlcTask Inputs/IO.st050_Mould_IO.stIn/aFromEngelRaw @bit 328 <-> IO Inputs/Var 7863
//     PlcTask Inputs/IO.st050_Mould_IO.stIn/aFromEngelRaw @bit 329 <-> IO Inputs/Var 7864
//     PlcTask Inputs/IO.st050_Mould_IO.stIn/aFromEngelRaw @bit 330 <-> IO Inputs/Var 7865
//     PlcTask Inputs/IO.st050_Mould_IO.stIn/aFromEngelRaw @bit 331 <-> IO Inputs/Var 7866
//     PlcTask Inputs/IO.st050_Mould_IO.stIn/aFromEngelRaw @bit 332 <-> IO Inputs/Var 7867
//     PlcTask Inputs/IO.st050_Mould_IO.stIn/aFromEngelRaw @bit 333 <-> IO Inputs/Var 7868
//     PlcTask Inputs/IO.st050_Mould_IO.stIn/aFromEngelRaw @bit 334 <-> IO Inputs/Var 7869
//     PlcTask Inputs/IO.st050_Mould_IO.stIn/aFromEngelRaw @bit 335 <-> IO Inputs/Var 7870
//     PlcTask Outputs/IO.st050_Mould_IO.stOut/aToEngelRaw <-> IO Outputs/Var 7824
//     PlcTask Outputs/IO.st050_Mould_IO.stOut/aToEngelRaw @bit 16 <-> IO Outputs/Var 7825
//     PlcTask Outputs/IO.st050_Mould_IO.stOut/aToEngelRaw @bit 32 <-> IO Outputs/Var 7826
//     PlcTask Outputs/IO.st050_Mould_IO.stOut/aToEngelRaw @bit 33 <-> IO Outputs/Var 7827
//     PlcTask Outputs/IO.st050_Mould_IO.stOut/aToEngelRaw @bit 34 <-> IO Outputs/Var 7828
//     PlcTask Outputs/IO.st050_Mould_IO.stOut/aToEngelRaw @bit 35 <-> IO Outputs/Var 7829
//     PlcTask Outputs/IO.st050_Mould_IO.stOut/aToEngelRaw @bit 36 <-> IO Outputs/Var 7830
//     PlcTask Outputs/IO.st050_Mould_IO.stOut/aToEngelRaw @bit 37 <-> IO Outputs/Var 7831
//     PlcTask Outputs/IO.st050_Mould_IO.stOut/aToEngelRaw @bit 38 <-> IO Outputs/Var 7832
//     PlcTask Outputs/IO.st050_Mould_IO.stOut/aToEngelRaw @bit 39 <-> IO Outputs/Var 7833
//     PlcTask Outputs/IO.st050_Mould_IO.stOut/aToEngelRaw @bit 40 <-> IO Outputs/Var 7834
//     PlcTask Outputs/IO.st050_Mould_IO.stOut/aToEngelRaw @bit 41 <-> IO Outputs/Var 7835
//     PlcTask Outputs/IO.st050_Mould_IO.stOut/aToEngelRaw @bit 42 <-> IO Outputs/Var 7836
//     PlcTask Outputs/IO.st050_Mould_IO.stOut/aToEngelRaw @bit 43 <-> IO Outputs/Var 7837
//     PlcTask Outputs/IO.st050_Mould_IO.stOut/aToEngelRaw @bit 44 <-> IO Outputs/Var 7838
//     PlcTask Outputs/IO.st050_Mould_IO.stOut/aToEngelRaw @bit 45 <-> IO Outputs/Var 7839
//     PlcTask Outputs/IO.st050_Mould_IO.stOut/aToEngelRaw @bit 46 <-> IO Outputs/Var 7840
//     PlcTask Outputs/IO.st050_Mould_IO.stOut/aToEngelRaw @bit 47 <-> IO Outputs/Var 7841
//     PlcTask Outputs/IO.st050_Mould_IO.stOut/aToEngelRaw @bit 48 <-> IO Outputs/Var 7842
//     PlcTask Outputs/IO.st050_Mould_IO.stOut/aToEngelRaw @bit 49 <-> IO Outputs/Var 7843
//     PlcTask Outputs/IO.st050_Mould_IO.stOut/aToEngelRaw @bit 50 <-> IO Outputs/Var 7844
//     PlcTask Outputs/IO.st050_Mould_IO.stOut/aToEngelRaw @bit 51 <-> IO Outputs/Var 7845
//     PlcTask Outputs/IO.st050_Mould_IO.stOut/aToEngelRaw @bit 52 <-> IO Outputs/Var 7846
//     PlcTask Outputs/IO.st050_Mould_IO.stOut/aToEngelRaw @bit 53 <-> IO Outputs/Var 7847
//     PlcTask Outputs/IO.st050_Mould_IO.stOut/aToEngelRaw @bit 54 <-> IO Outputs/Var 7848
//     PlcTask Outputs/IO.st050_Mould_IO.stOut/aToEngelRaw @bit 55 <-> IO Outputs/Var 7849
//     PlcTask Outputs/IO.st050_Mould_IO.stOut/aToEngelRaw @bit 56 <-> IO Outputs/Var 7850
//     PlcTask Outputs/IO.st050_Mould_IO.stOut/aToEngelRaw @bit 72 <-> IO Outputs/Var 7851
//     PlcTask Outputs/IO.st050_Mould_IO.stOut/aToEngelRaw @bit 88 <-> IO Outputs/Var 7852
//     PlcTask Outputs/IO.st050_Mould_IO.stOut/aToEngelRaw @bit 104 <-> IO Outputs/Var 7853
//     PlcTask Outputs/IO.st050_Mould_IO.stOut/aToEngelRaw @bit 120 <-> IO Outputs/Var 7854
//     PlcTask Outputs/IO.st050_Mould_IO.stOut/aToEngelRaw @bit 136 <-> IO Outputs/Var 7855
//     PlcTask Outputs/IO.st050_Mould_IO.stOut/aToEngelRaw @bit 152 <-> IO Outputs/Var 7856
//     PlcTask Outputs/IO.st050_Mould_IO.stOut/aToEngelRaw @bit 168 <-> IO Outputs/Var 7857
//     PlcTask Outputs/IO.st050_Mould_IO.stOut/aToEngelRaw @bit 184 <-> IO Outputs/Var 7858
//     PlcTask Outputs/IO.st050_Mould_IO.stOut/aToEngelRaw @bit 200 <-> IO Outputs/Var 7859
//     PlcTask Outputs/IO.st050_Mould_IO.stOut/aToEngelRaw @bit 216 <-> IO Outputs/Var 7860
//     PlcTask Outputs/IO.st050_Mould_IO.stOut/aToEngelRaw @bit 232 <-> IO Outputs/Var 7861
//     PlcTask Outputs/IO.st050_Mould_IO.stOut/aToEngelRaw @bit 248 <-> IO Outputs/Var 7862
//     PlcTask Outputs/IO.st050_Mould_IO.stOut/aToEngelRaw @bit 264 <-> IO Outputs/Var 7863
//     PlcTask Outputs/IO.st050_Mould_IO.stOut/aToEngelRaw @bit 280 <-> IO Outputs/Var 7864
//     PlcTask Outputs/IO.st050_Mould_IO.stOut/aToEngelRaw @bit 296 <-> IO Outputs/Var 7865
//     PlcTask Outputs/IO.st050_Mould_IO.stOut/aToEngelRaw @bit 312 <-> IO Outputs/Var 7866
//     PlcTask Outputs/IO.st050_Mould_IO.stOut/aToEngelRaw @bit 328 <-> IO Outputs/Var 7867
//     PlcTask Outputs/IO.st050_Mould_IO.stOut/aToEngelRaw @bit 329 <-> IO Outputs/Var 7868
//     PlcTask Outputs/IO.st050_Mould_IO.stOut/aToEngelRaw @bit 330 <-> IO Outputs/Var 7869
//     PlcTask Outputs/IO.st050_Mould_IO.stOut/aToEngelRaw @bit 331 <-> IO Outputs/Var 7870
//     PlcTask Outputs/IO.st050_Mould_IO.stOut/aToEngelRaw @bit 332 <-> IO Outputs/Var 7871
//     PlcTask Outputs/IO.st050_Mould_IO.stOut/aToEngelRaw @bit 333 <-> IO Outputs/Var 7872
//     PlcTask Outputs/IO.st050_Mould_IO.stOut/aToEngelRaw @bit 334 <-> IO Outputs/Var 7873
//     PlcTask Outputs/IO.st050_Mould_IO.stOut/aToEngelRaw @bit 335 <-> IO Outputs/Var 7921
//   PLC/PLC Instance <-> Device 3 (EtherCAT)/Term 1 (EK1100)/Storage|Casting (EK1122)/Storage (EK1100)
//     PlcTask Inputs/IO.stControlCabinetIO.stIn/IarrEcStates[3] <-> InfoData/State
//   PLC/PLC Instance <-> Device 3 (EtherCAT)/Term 1 (EK1100)/Term 33 (EL6910)
//     PlcTask Inputs/IO.stSafetyIO.stIn/bSAFE_Area_Ok_ST10 <-> StandardInputs/SafetyGates.Safe_A_73
//     PlcTask Inputs/IO.stSafetyIO.stIn/bSAFE_Area_Ok_ST20 <-> StandardInputs/SafetyGates.Safe_B_74
//     PlcTask Inputs/IO.stSafetyIO.stIn/bSAFE_Areas_Ok <-> StandardInputs/SafetyGates.Safe_Area_137
//     PlcTask Inputs/IO.stSafetyIO.stIn/bSAFE_DRIVES_HG_STO <-> StandardInputs/Rackfeeder_Axis.STO_Active_84
//     PlcTask Inputs/IO.stSafetyIO.stIn/bSAFE_DRIVE_A_STO <-> StandardInputs/Oven_Axis.STO_Active_OvenA_94
//     PlcTask Inputs/IO.stSafetyIO.stIn/bSAFE_DRIVE_B_STO <-> StandardInputs/Oven_Axis.STO_Active_OvenB_127
//     PlcTask Inputs/IO.stSafetyIO.stIn/bSAFE_ES_Ok <-> StandardInputs/TwinSafeMain.Safe_62
//     PlcTask Inputs/IO.stSafetyIO.stIn/bSAFE_EStop_State[1] <-> StandardInputs/TwinSafeMain.Emergency01_Active_63
//     PlcTask Inputs/IO.stSafetyIO.stIn/bSAFE_EStop_State[2] <-> StandardInputs/TwinSafeMain.Emergency02_Active_64
//     PlcTask Inputs/IO.stSafetyIO.stIn/bSafe_ComError_Master[1] <-> StandardInputs/TwinSafeMain.ComErr_99
//     PlcTask Inputs/IO.stSafetyIO.stIn/bSafe_EL6900_WcState[0] <-> WcState/WcState
//     PlcTask Inputs/IO.stSafetyIO.stIn/bSafe_FbError_Master[1] <-> StandardInputs/TwinSafeMain.FBErr_98
//     PlcTask Inputs/IO.stSafetyIO.stIn/bSafe_OtherError_Master[1] <-> StandardInputs/TwinSafeMain.OtherErr_56
//     PlcTask Inputs/IO.stSafetyIO.stIn/bSafe_OutError_Master[1] <-> StandardInputs/TwinSafeMain.OutErr_101
//     PlcTask Inputs/Safety.arrSaftyDoors[0].stHwIn/tsOpen <-> StandardInputs/SafetyGates.Door_Open_A_75
//     PlcTask Inputs/Safety.arrSaftyDoors[0].stHwIn/tsSafe <-> StandardInputs/SafetyGates.Safe_A_73
//     PlcTask Inputs/Safety.arrSaftyDoors[0].stHwIn/tsSegment_Open <-> StandardInputs/SafetyGates.Segment_Open_A_132
//     PlcTask Inputs/Safety.arrSaftyDoors[1].stHwIn/tsOpen <-> StandardInputs/SafetyGates.Door_Open_B_76
//     PlcTask Inputs/Safety.arrSaftyDoors[1].stHwIn/tsSafe <-> StandardInputs/SafetyGates.Safe_B_74
//     PlcTask Inputs/Safety.arrSaftyDoors[1].stHwIn/tsSegment_Open <-> StandardInputs/SafetyGates.Segment_Open_B_133
//     PlcTask Outputs/IO.stSafetyIO.stOut/bRestartPLC <-> StandardOutputs/TwinSafeMain.Restart_61
//     PlcTask Outputs/IO.stSafetyIO.stOut/bSafe_Tsg_Run[1] <-> StandardOutputs/TwinSafeMain.RunStop_54
//     PlcTask Outputs/IO.stSafetyIO.stOut/bSafetyErrAck[1] <-> StandardOutputs/Oven_Axis.Error_Ack_OvenA_122
//     PlcTask Outputs/IO.stSafetyIO.stOut/bSafetyErrAck[1] <-> StandardOutputs/Oven_Axis.Error_Ack_OvenB_88
//     PlcTask Outputs/IO.stSafetyIO.stOut/bSafetyErrAck[1] <-> StandardOutputs/Rackfeeder_Axis.Error_Ack_80
//     PlcTask Outputs/IO.stSafetyIO.stOut/bSafetyErrAck[1] <-> StandardOutputs/TwinSafeMain.DriveRestart_117
//     PlcTask Outputs/IO.stSafetyIO.stOut/bSafetyErrAck[1] <-> StandardOutputs/TwinSafeMain.ErrAck_53
//     PlcTask Outputs/Safety.arrSaftyDoors[0].stHwOut/tsLockCmd <-> StandardOutputs/SafetyGates.LockCmd_A_109
//     PlcTask Outputs/Safety.arrSaftyDoors[0].stHwOut/tsRestart <-> StandardOutputs/SafetyGates.Restart_A_71
//     PlcTask Outputs/Safety.arrSaftyDoors[1].stHwOut/tsLockCmd <-> StandardOutputs/SafetyGates.LockCmd_B_110
//     PlcTask Outputs/Safety.arrSaftyDoors[1].stHwOut/tsRestart <-> StandardOutputs/SafetyGates.Restart_B_72
//   PLC/PLC Instance <-> Device 3 (EtherCAT)/Term 1 (EK1100)/Term 5 (EL1104)
//     PlcTaskFast Inputs/IO.st030_Handling_IO.stIn/bRefposX <-> Channel 1/bRefposX
//   PLC/PLC Instance <-> Device 3 (EtherCAT)/Term 1 (EK1100)/Term 7 (EL6224)
//     PlcTask Inputs/GVL_BVS_Sensor.BVS_IolState <-> DeviceState Inputs/State Ch4
//     PlcTask Inputs/GVL_BVS_Sensor.BVS_Sensor_IN @bit {24..240 step 8} <-> IO-Link Port4_in/Data Byte {0..27}  (28 links)
//     PlcTask Inputs/GVL_BVS_Sensor.BVS_Sensor_IN @bit 7 <-> IO-Link Port4_in/Device Locked
//     PlcTask Inputs/GVL_BVS_Sensor.BVS_Sensor_IN @bit 12 <-> IO-Link Port4_in/Input Data Error
//     PlcTask Inputs/GVL_BVS_Sensor.BVS_Sensor_IN @bit 18 <-> IO-Link Port4_in/Job End
//     PlcTask Inputs/GVL_BVS_Sensor.BVS_Sensor_IN @bit 250 <-> IO-Link Port4_in/Job End_1
//     PlcTask Inputs/GVL_BVS_Sensor.BVS_Sensor_IN @bit 19 <-> IO-Link Port4_in/Job Error
//     PlcTask Inputs/GVL_BVS_Sensor.BVS_Sensor_IN @bit 251 <-> IO-Link Port4_in/Job Error_1
//     PlcTask Inputs/GVL_BVS_Sensor.BVS_Sensor_IN @bit 17 <-> IO-Link Port4_in/Job Start
//     PlcTask Inputs/GVL_BVS_Sensor.BVS_Sensor_IN @bit 249 <-> IO-Link Port4_in/Job Start_1
//     PlcTask Inputs/GVL_BVS_Sensor.BVS_Sensor_IN @bit 5 <-> IO-Link Port4_in/Ready
//     PlcTask Inputs/GVL_BVS_Sensor.BVS_Sensor_IN @bit 10 <-> IO-Link Port4_in/Report Error
//     PlcTask Inputs/GVL_BVS_Sensor.BVS_Sensor_IN @bit 1 <-> IO-Link Port4_in/Result Data Available
//     PlcTask Inputs/GVL_BVS_Sensor.BVS_Sensor_IN @bit 9 <-> IO-Link Port4_in/Result Data Error
//     PlcTask Inputs/GVL_BVS_Sensor.BVS_Sensor_IN @bit 3 <-> IO-Link Port4_in/Simulation Mode
//     PlcTask Inputs/GVL_BVS_Sensor.BVS_Sensor_IN @bit 15 <-> IO-Link Port4_in/System Error
//     PlcTask Inputs/GVL_BVS_Sensor.BVS_Sensor_IN @bit 21 <-> IO-Link Port4_in/Toggle Out
//     PlcTask Inputs/GVL_BVS_Sensor.BVS_Sensor_IN @bit 253 <-> IO-Link Port4_in/Toggle Out_1
//     PlcTask Inputs/GVL_BVS_Sensor.BVS_Sensor_IN @bit 8 <-> IO-Link Port4_in/Trigger Overflow
//     PlcTask Inputs/GVL_BVS_Sensor.BVS_Sensor_IN <-> IO-Link Port4_in/Waiting For Trigger
//     PlcTask Outputs/GVL_BVS_Sensor.BVS_Sensor_Out @bit {8..240 step 8} <-> IO-Link Port4_out/Data Byte {0..29}  (30 links)
//     PlcTask Outputs/GVL_BVS_Sensor.BVS_Sensor_Out <-> IO-Link Port4_out/Job
//     PlcTask Outputs/GVL_BVS_Sensor.BVS_Sensor_Out @bit 248 <-> IO-Link Port4_out/Job_1
//     PlcTask Outputs/GVL_BVS_Sensor.BVS_Sensor_Out @bit 2 <-> IO-Link Port4_out/Reset Error
//     PlcTask Outputs/GVL_BVS_Sensor.BVS_Sensor_Out @bit 250 <-> IO-Link Port4_out/Reset Error_1
//     PlcTask Outputs/GVL_BVS_Sensor.BVS_Sensor_Out @bit 6 <-> IO-Link Port4_out/Toggle In
//     PlcTask Outputs/GVL_BVS_Sensor.BVS_Sensor_Out @bit 254 <-> IO-Link Port4_out/Toggle In_1
//     PlcTask Outputs/GVL_BVS_Sensor.BVS_Sensor_Out @bit 1 <-> IO-Link Port4_out/Trigger
//     PlcTask Outputs/GVL_BVS_Sensor.BVS_Sensor_Out @bit 249 <-> IO-Link Port4_out/Trigger_1
//     PlcTaskFast Inputs/IO.st030_Handling_IO.stIn/bRefposY <-> Beckhoff IO Box_IN/bRefposY
//     PlcTaskFast Inputs/IO.st030_Handling_IO.stIn/bRefposZ <-> Beckhoff IO Box_IN/bRefposZ
//     PlcTaskFast Inputs/IO.st030_Handling_IO.stIn/fMeasurementA <-> IO-Link Port2_in/Measurement value: Distance
//     PlcTaskFast Inputs/IO.st030_Handling_IO.stIn/fMeasurementB <-> IO-Link Port3_in/Measurement value: Distance
//   PLC/PLC Instance <-> Device 3 (EtherCAT)/Term 1 (EK1100)/Term 71 (EL1008)
//     PlcTask Inputs/HMI.stHmiHw.stIn.stP51A_S1HandBs/bDistance <-> Channel 8/Input_distance
//     PlcTask Inputs/HMI.stHmiHw.stIn.stP51A_S1HandBs/bJog <-> Channel 7/Input_jog
//     PlcTask Inputs/HMI.stHmiHw.stIn.stP51A_S1HandBs/bSelect01 <-> Channel 1/Input_01
//     PlcTask Inputs/HMI.stHmiHw.stIn.stP51A_S1HandBs/bSelect02 <-> Channel 2/Input_02
//     PlcTask Inputs/HMI.stHmiHw.stIn.stP51A_S1HandBs/bSelect03 <-> Channel 3/Input_03
//     PlcTask Inputs/HMI.stHmiHw.stIn.stP51A_S1HandBs/bSelect04 <-> Channel 4/Input_04
//     PlcTask Inputs/HMI.stHmiHw.stIn.stP51A_S1HandBs/bSelect05 <-> Channel 5/Input_05
//     PlcTask Inputs/HMI.stHmiHw.stIn.stP51A_S1HandBs/bSelect06 <-> Channel 6/Input_06
//   PLC/PLC Instance <-> Device 3 (EtherCAT)/Term 1 (EK1100)/Term 73 (EL1008)
//     PlcTask Inputs/HMI.stHmiHw.stIn.stP51A_S1HandBs/bAlt <-> Channel 5/Input_alt
//     PlcTask Inputs/HMI.stHmiHw.stIn.stP51A_S1HandBs/bDown <-> Channel 1/Input_down
//     PlcTask Inputs/HMI.stHmiHw.stIn.stP51A_S1HandBs/bLeft <-> Channel 4/Input_left
//     PlcTask Inputs/HMI.stHmiHw.stIn.stP51A_S1HandBs/bReset <-> Channel 2/Input_reset
//     PlcTask Inputs/HMI.stHmiHw.stIn.stP51A_S1HandBs/bRight <-> Channel 6/Input_right
//     PlcTask Inputs/HMI.stHmiHw.stIn.stP51A_S1HandBs/bUp <-> Channel 3/Input_up
//   PLC/PLC Instance <-> Device 3 (EtherCAT)/Term 1 (EK1100)/Term 74 (EL2008)
//     PlcTask Outputs/HMI.stHmiHw.stOut.stP51A_S1HandBs/bLedDistance <-> Channel 8/Output_distance
//     PlcTask Outputs/HMI.stHmiHw.stOut.stP51A_S1HandBs/bLedLeft <-> Channel 7/Output_left
//     PlcTask Outputs/HMI.stHmiHw.stOut.stP51A_S1HandBs/bLedSelect01 <-> Channel 1/Output_01
//     PlcTask Outputs/HMI.stHmiHw.stOut.stP51A_S1HandBs/bLedSelect02 <-> Channel 2/Output_02
//     PlcTask Outputs/HMI.stHmiHw.stOut.stP51A_S1HandBs/bLedSelect03 <-> Channel 3/Output_03
//     PlcTask Outputs/HMI.stHmiHw.stOut.stP51A_S1HandBs/bLedSelect04 <-> Channel 4/Output_04
//     PlcTask Outputs/HMI.stHmiHw.stOut.stP51A_S1HandBs/bLedSelect05 <-> Channel 5/Output_05
//     PlcTask Outputs/HMI.stHmiHw.stOut.stP51A_S1HandBs/bLedSelect06 <-> Channel 6/Output_06
//   PLC/PLC Instance <-> Device 3 (EtherCAT)/Term 1 (EK1100)/Term 75 (EL2008)
//     PlcTask Outputs/HMI.stHmiHw.stOut.stP51A_S1HandBs/bLedAlt <-> Channel 3/Output_alt
//     PlcTask Outputs/HMI.stHmiHw.stOut.stP51A_S1HandBs/bLedDown <-> Channel 5/Output_down
//     PlcTask Outputs/HMI.stHmiHw.stOut.stP51A_S1HandBs/bLedJog <-> Channel 2/Output_jog
//     PlcTask Outputs/HMI.stHmiHw.stOut.stP51A_S1HandBs/bLedRight <-> Channel 4/Output_right
//     PlcTask Outputs/HMI.stHmiHw.stOut.stP51A_S1HandBs/bLedUp <-> Channel 1/Output_up
//   PLC/PLC Instance <-> NC-Task 1 SAF/Axes/Oven A
//     PlcTask Inputs/NcIO.stAxis_ST010_OvenA.NcToPlc <-> Outputs/ToPlc
//     PlcTask Outputs/NcIO.stAxis_ST010_OvenA.PlcToNc <-> Inputs/FromPlc
//   PLC/PLC Instance <-> NC-Task 1 SAF/Axes/Oven A CH1
//     PlcTask Inputs/NcIO.stAxis_ST010_OvenACh1.NcToPlc <-> Outputs/ToPlc
//     PlcTask Outputs/NcIO.stAxis_ST010_OvenACh1.PlcToNc <-> Inputs/FromPlc
//   PLC/PLC Instance <-> NC-Task 1 SAF/Axes/Oven A CH2
//     PlcTask Inputs/NcIO.stAxis_ST010_OvenACh2.NcToPlc <-> Outputs/ToPlc
//     PlcTask Outputs/NcIO.stAxis_ST010_OvenACh2.PlcToNc <-> Inputs/FromPlc
//   PLC/PLC Instance <-> NC-Task 1 SAF/Axes/Oven B
//     PlcTask Inputs/NcIO.stAxis_ST020_OvenB.NcToPlc <-> Outputs/ToPlc
//     PlcTask Outputs/NcIO.stAxis_ST020_OvenB.PlcToNc <-> Inputs/FromPlc
//   PLC/PLC Instance <-> NC-Task 1 SAF/Axes/Oven B CH1
//     PlcTask Inputs/NcIO.stAxis_ST020_OvenBCh1.NcToPlc <-> Outputs/ToPlc
//     PlcTask Outputs/NcIO.stAxis_ST020_OvenBCh1.PlcToNc <-> Inputs/FromPlc
//   PLC/PLC Instance <-> NC-Task 1 SAF/Axes/Oven B CH2
//     PlcTask Inputs/NcIO.stAxis_ST020_OvenBCh2.NcToPlc <-> Outputs/ToPlc
//     PlcTask Outputs/NcIO.stAxis_ST020_OvenBCh2.PlcToNc <-> Inputs/FromPlc
//   PLC/PLC Instance <-> NC-Task 1 SAF/Axes/Rackfeeder X
//     PlcTask Inputs/NcIO.stAxis_ST030_AxisX.NcToPlc <-> Outputs/ToPlc
//     PlcTask Outputs/NcIO.stAxis_ST030_AxisX.PlcToNc <-> Inputs/FromPlc
//   PLC/PLC Instance <-> NC-Task 1 SAF/Axes/Rackfeeder Y
//     PlcTask Inputs/NcIO.stAxis_ST030_AxisY.NcToPlc <-> Outputs/ToPlc
//     PlcTask Outputs/NcIO.stAxis_ST030_AxisY.PlcToNc <-> Inputs/FromPlc
//   PLC/PLC Instance <-> NC-Task 1 SAF/Axes/Rackfeeder Z
//     PlcTask Inputs/NcIO.stAxis_ST030_AxisZ.NcToPlc <-> Outputs/ToPlc
//     PlcTask Outputs/NcIO.stAxis_ST030_AxisZ.PlcToNc <-> Inputs/FromPlc
//   PLC/PLC Instance <-> NC-Task 1 SAF/Axes/Storage A
//     PlcTask Inputs/NcIO.stAxis_ST040_Axis1.NcToPlc <-> Outputs/ToPlc
//     PlcTask Outputs/NcIO.stAxis_ST040_Axis1.PlcToNc <-> Inputs/FromPlc
//   PLC/PLC Instance <-> NC-Task 1 SAF/Axes/Storage B
//     PlcTask Inputs/NcIO.stAxis_ST040_Axis2.NcToPlc <-> Outputs/ToPlc
//     PlcTask Outputs/NcIO.stAxis_ST040_Axis2.PlcToNc <-> Inputs/FromPlc

CONFIGURATION PLC
    RESOURCE PLC ON TwinCAT3
        TASK PlcTask(INTERVAL := T#5ms, PRIORITY := 10);
        TASK PlcTaskFast(INTERVAL := T#1ms, PRIORITY := 4);
        PROGRAM MAIN WITH PlcTask : MAIN;
        PROGRAM MAIN_Fast WITH PlcTaskFast : MAIN_Fast;
    END_RESOURCE
END_CONFIGURATION

// ---- Background/UnitTest/Enumerations/E_TestCaseState.TcDUT
/// Enumeration of all possible test case states
TYPE E_TestCaseState :
(
	/// Test case state not set
	eTestCaseState_none := 0,
	/// Test case ready
	eTestCaseState_ready,
	/// Test case is running
	eTestCaseState_running,
	/// Test case finished
	eTestCaseState_finished,
	/// Test case error (execution error)
	eTestCaseState_error
);
END_TYPE

// ---- Background/UnitTest/Enumerations/E_TestResult.TcDUT
/// Enumeration of all possible test case states
TYPE E_TestResult :
(
	/// Test result not set
	eTestResult_none := 0,
	/// Test result ok
	eTestResult_ok,
	/// Test result not ok
	eTestResult_nok
);
END_TYPE

// ---- Background/UnitTest/TestCases/StationTest/Structures/ST_TestStation_IN.TcDUT
TYPE ST_TestStation_IN :
STRUCT
	bTestInput	: BOOL;
END_STRUCT
END_TYPE

// ---- Background/UnitTest/TestCases/StationTest/Structures/ST_TestStation_IO.TcDUT
TYPE ST_TestStation_IO :
STRUCT
	stIn	: ST_TestStation_IN;
	stOut	: ST_TestStation_OUT;
END_STRUCT
END_TYPE

// ---- Background/UnitTest/TestCases/StationTest/Structures/ST_TestStation_OUT.TcDUT
TYPE ST_TestStation_OUT :
STRUCT
	bTestInput	: BOOL;
END_STRUCT
END_TYPE

// ---- DUTs/Configuration/ST_Configuration.TcDUT
TYPE ST_Configuration :
STRUCT
	/// debug logging configuration
	stLogConfig			: ST_LoggingConfig;
	
	stVar2FileConfig	: ST_Var2File_Config;
END_STRUCT
END_TYPE

// ---- POUs/Components/AxisDriver/Enumerations/E_Axis.TcDUT
/// Enumeration of all axis drives.
TYPE E_Axis :
(
	eAxis_none := 0,
	// UnitTest axis
	
	// oven B CH
	eAxis_OvenB_CH1,
	eAxis_OvenB_CH2,
	
	// handling
	eAxis_Handling_X,
	eAxis_Handling_Y,
	eAxis_Handling_Z,
	
	// oven B A
	eAxis_OvenB,
	eAxis_OvenA,
	
	// oven A CH
	eAxis_OvenA_CH1,
	eAxis_OvenA_CH2,

	// storage
	eAxis_Storage1,
	eAxis_Storage2,
	
	eAxis_MaxAxis
);
END_TYPE

// ---- POUs/Components/AxisDriver/Enumerations/E_GearMode.TcDUT
/// Enumeration of possible axis gear modes.
TYPE E_GearMode :
(
	/// Gear mode not set
	eGearMode_none := 0,
	/// Gear in
	eGearMode_in,
	/// Gear out
	eGearMode_out
);
END_TYPE

// ---- POUs/Components/AxisDriver/Enumerations/E_JogDirection.TcDUT
/// Enumeration of possible jog directions.
TYPE E_JogDirection :
(
	/// Jog direction not set
	eJogDirection_none := 0,
	/// Jog direction positive
	eJogDirection_pos,
	/// Jog direction negative
	eJogDirection_neg
);
END_TYPE

// ---- POUs/Components/AxisDriver/Enumerations/E_ManualMode.TcDUT
/// Enumeration of possible jog modi.
TYPE E_ManualMode :
(
	/// Manual mode - Tippen konstant
	eManualMode_Tippen := 0,
	
	/// Manual mode - Sollposition Absolut
	//eManualMode_MoveSollAbs,
	/// Manual mode - Relativ 0.01 Einheit
	eManualMode_Jog001,	
	/// Manual mode - Relativ 0.1 Einheit
	eManualMode_Jog01,
	/// Manual mode - Relativ 1 Einheit
	eManualMode_Jog1,
	/// Manual mode - Relativ 10 Einheiten
	eManualMode_Jog10,
	/// Manual mode - Relativ 100 Einheiten
	eManualMode_Jog100,
	/// Manual mode not set
	eManualMode_none
);
END_TYPE

// ---- POUs/Components/AxisDriver/Enumerations/E_MotionCommand.TcDUT
/// Enumeration of possible axis motion commands.
TYPE E_MotionCommand :
(
	/// No command
	eMotionCommand_none := 0,
	/// Reset axis
	eMotionCommand_reset := 1,
	/// Axis halt (default stopping method)
	eMotionCommand_halt := 2,
	/// Axis stop (needs reset before next motion command)
	eMotionCommand_stop := 3,
	/// Axis homing
	eMotionCommand_home := 4,
	/// Set axis position
	eMotionCommand_setPos := 5,
	/// Jog axis
	eMotionCommand_jog := 6,
	/// Jog axis accelerating
	eMotionCommand_jogAcc := 7,
	/// Move axis to point
	eMotionCommand_moveAbs := 8,
	/// Move axis additive
	eMotionCommand_moveAdd := 9,
	/// Move axis relative
	eMotionCommand_moveRel := 10,
	/// Move axis modulo
	eMotionCommand_moveMod := 11,
	/// Move axis velocity (endles)
	eMotionCommand_moveVel := 12,
	/// Apply axis torque
	eMotionCommand_torque := 13,
	/// Gear axis in (electronic) or change gear ratio
	eMotionCommand_gearIn := 14,
	/// Gear axis out (electronic), default behavior: halt axis after gear out
	eMotionCommand_gearOut := 15,
	/// Axis start/stop touch probe
	eMotionCommand_touchProbe := 16,
	/// Force MC reset axis
	eMotionCommand_resetMc := 17,
	/// Group add
	eMotionCommand_GroupAdd := 18,
	/// torque control
	eMotionCommand_torqCtrl := 19,
	
	/// set ax axis position offset
	eMotionCommand_setAxPosOffs := 20
);
END_TYPE

// ---- POUs/Components/AxisDriver/Enumerations/E_Mover_XTS.TcDUT
//{attribute 'qualified_only'}
//{attribute 'strict'}
TYPE E_Mover_XTS :
(
	eMoverXts_none := 0,
	// UnitTest axis
	eMoverXts_01,
	eMoverXts_02,
	eMoverXts_03,
	eMoverXts_04,
	eMoverXts_05,
	eMoverXts_06,
	eMoverXts_07,
	eMoverXts_08,
	eMoverXts_09,
	eMoverXts_10,
	eMoverXts_11,
	eMoverXts_12,
	eMoverXts_13,
	eMoverXts_14,
	eMoverXts_15,
	eMoverXts_16,
	eMoverXts_17,
	eMoverXts_18,
	eMoverXts_19,
	eMoverXts_20,
	eMoverXts_21,
	eMoverXts_22,
	eMoverXts_23,
	eMoverXts_24,
	eMoverXts_25,
	eMoverXts_26,
	
	eMoverXts_MaxAxis
);
END_TYPE

// ---- POUs/Components/AxisDriver/Enumerations/E_SoECommand.TcDUT
/// SoE commands
TYPE E_SoECommand :
(
	eSoECommand_none := 0,
	eSoECommand_writeIndraDrvPos
);
END_TYPE

// ---- POUs/Components/AxisDriver/Structures/AdditionalAxisIO/ST_AxisIn.TcDUT
TYPE ST_AxisIn :
STRUCT
	/// Ec Box State
	iEcState				: UINT;
	/// Motortemp: [1/10 °C]
	iMotorTemperature		: INT;
	/// Amplifiertemp: [1/10 °C]
	iAmplifierTemperature	: INT;
	/// Versorgungsspannung
	iActualMainVoltage		: INT;
	/// User Status Wort
	nUserStateWord			: WORD;
END_STRUCT
END_TYPE

// ---- POUs/Components/AxisDriver/Structures/AdditionalAxisIO/ST_AxisIO.TcDUT
/// Additional axis IO (direct linked) for AX5xxx axis.
TYPE ST_AxisIO :
STRUCT
	stIn 	AT %I* 	:ST_AxisIn;
	stOut	AT %Q* 	:ST_AxisOut;
END_STRUCT
END_TYPE

// ---- POUs/Components/AxisDriver/Structures/AdditionalAxisIO/ST_AxisOut.TcDUT
TYPE ST_AxisOut :
STRUCT
	/// Ext. fan control
	bExternalFan: BOOL;
	/// The bipolar torque limit value limits the maximum torque symmetrically in both directions. [1/10 %]
	iBipolarTorqueLimitValue: INT := 4000;
	/// During the torque control operation mode of the drive, torque command values are transferred from the control unit to the drive. [1/10 %]
	iTorqueCommandValue: INT;
	/// This value is added as an offset to the torque command value. [1/10 %]
	iAdditiveTorqueCommandValue: INT;
END_STRUCT
END_TYPE

// ---- POUs/Components/AxisDriver/Structures/AdditionalAxisIO/ST_AxisVirtualIO.TcDUT
/// Dummy IO for virtual axis.
TYPE ST_AxisVirtualIO :
STRUCT
	stIn: ST_AxisIn;
	stOut: ST_AxisOut;
END_STRUCT
END_TYPE

// ---- POUs/Components/AxisDriver/Structures/SoE/ST_AxisSoE.TcDUT
TYPE ST_AxisSoE :
STRUCT
	// command
	eCmd		: E_SoECommand;
	
	// SoE FB's 
	fbSoEWrite	: FB_SoEWrite;
	fbSoECmd 	: FB_SoEExecuteCommand;
	
	// helper var's
	nStep		: INT;
	fRealValue	: REAL;
END_STRUCT
END_TYPE

// ---- POUs/Components/AxisDriver/Structures/ST_AxisDriverParameter.TcDUT
/// Parameter set for axis driver
TYPE ST_AxisDriverParameter :
STRUCT
	/// General axis parameter
	stGeneralPrm: ST_AxisGeneralParameter;
	/// Parameter for halting the axis
	stHaltPrm: ST_AxisHaltParameter;
	/// Parameter for stopping the axis
	stStopPrm: ST_AxisStopParameter;
	/// Parameter for axis homing
	stHomingPrm: ST_AxisHomingParameter;
	/// Parameter for axis set position
	stSetPosPrm: ST_AxisSetPosParameter;
	/// Parameter for axis homing
	stJogPrm: ST_AxisJogParameter;
	/// Parameter for accelerating jog
	stJogAccPrm: ST_AxisJogAccParameter;
	/// Parameter for move axis absolute
	stMovAbsPrm: ST_AxisMoveAbsParameter;
	/// Parameter for move axis additive
	stMovAddPrm: ST_AxisMoveAddParameter;
	/// Parameter for move axis relative
	stMovRelPrm: ST_AxisMoveRelParameter;
	/// Parameter for move axis modulo
	stMovModPrm: ST_AxisMoveModParameter;
	/// Parameter for move axis velocity
	stMovVelPrm: ST_AxisMoveVelParameter;
	/// Parameter for axis electronic gear-in
	stGearInPrm: ST_AxisGearInParameter;
	/// Parameter for axis electronic gear-out
	stGearOutPrm: ST_AxisGearOutParameter;
	/// Parameter for axis torque control
	stTorqCtrlPrm: ST_AxisTorqCtrlParameter;
END_STRUCT
END_TYPE

// ---- POUs/Components/AxisDriver/Structures/ST_AxisGearInParameter.TcDUT
/// GearIn parameter strucure
TYPE ST_AxisGearInParameter :
STRUCT
	eMasterId: E_Axis;
	fbMaster: REFERENCE TO AXIS_REF;
	fGearRatio: LREAL;
	fAcceleration: LREAL;
	fDeceleration: LREAL;
	fJerk: LREAL;
	eBufferMode: MC_BufferMode;
	stOptions: ST_GearInDynOptions;
END_STRUCT
END_TYPE

// ---- POUs/Components/AxisDriver/Structures/ST_AxisGearOutParameter.TcDUT
/// GearOut parameter strucure
TYPE ST_AxisGearOutParameter :
STRUCT
	/// Halt axis after gear out
	bHaltAxis: BOOL := TRUE;
	/// Gear out (not implemented)
	stOptions: ST_GearOutOptions;
END_STRUCT
END_TYPE

// ---- POUs/Components/AxisDriver/Structures/ST_AxisManager.TcDUT
TYPE ST_AxisManager :
STRUCT
	// HMI page axis manager
	
	// info flags, pos & text
	bAxisEnabled,
	bCalibrated,
	bSetCalibrationVisible,
	bResetCalibrationVisible,
	bEnablePosSet 	: BOOL;
	
	fActPos 		: LREAL;
	stBmk, stName, 
	stUnit, stInfo 	: ST_Text;
	//----------
	
	// additional axis disable flag
	bDisable,
	// disable soft limits flag
	bDisableSoftLimits,
	
	// set/reset calibration flag (ax must have no error and enable)
	bSetCalibration,
	bResetCalibration,
	
	// use local calibration- or sxis calibration flag
	bUseLocalCalibration, // setting intern!
	
	// trigger to set position (ax not enabled)
	bSetPosGo 			: BOOL;
	// absolute position to set
	fSetPos 			: REAL;
END_STRUCT
END_TYPE

// ---- POUs/Components/AxisDriver/Structures/ST_AxisTorqCtrlParameter.TcDUT
/// Torque control parameter strucure
TYPE ST_AxisTorqCtrlParameter :
STRUCT
	fTorque				: LREAL;	// %
	fTorqueRamp			: LREAL;
    fVelocityLimitHigh	: LREAL;
    fVelocityLimitLow	: LREAL;
	bContinuousUpdate	: BOOL := TRUE;
	bRelative			: BOOL;
    eBufferMode			: MC_BufferMode;
	stOptions			: ST_TorqueControlOptions;
END_STRUCT
END_TYPE

// ---- POUs/Components/AxisDriver/Structures/ST_AxisGeneralParameter.TcDUT
/// General axis parameter set
TYPE ST_AxisGeneralParameter :
STRUCT
	/// Auto power off axis (economize)
	bEnableAutoPowerOff	: BOOL := FALSE;
	/// Delay time until power off idle axis
	tAutoPowerOffDelay	: TIME := TIME#10S0MS;
	/// Threshold temperature [1/10 °C] for external fan.
	iExtFanThreshold	: INT := 500;
	/// Factor for torque value
	fTorqueFactor		: REAL := 1;
END_STRUCT
END_TYPE

// ---- POUs/Components/AxisDriver/Structures/ST_AxisHaltParameter.TcDUT
TYPE ST_AxisHaltParameter EXTENDS ST_AxisStopParameter :
STRUCT
	eBufferMode: MC_BufferMode := MC_Aborting;
END_STRUCT
END_TYPE

// ---- POUs/Components/AxisDriver/Structures/ST_AxisHomingParameter.TcDUT
TYPE ST_AxisHomingParameter :
STRUCT
	bCalibrationCam: BOOL;
	fPosition: LREAL := DEFAULT_HOME_POSITION;
	eHomingMode: MC_HomingMode := MC_DefaultHoming;
	eBufferMode: MC_BufferMode := MC_Aborting;
	stOptions: ST_HomingOptions;
END_STRUCT
END_TYPE

// ---- POUs/Components/AxisDriver/Structures/ST_AxisJogAccParameter.TcDUT
/// Accelerating jog parameter strucure
TYPE ST_AxisJogAccParameter EXTENDS ST_AxisMoveParameter :
STRUCT
	/// Jog axis backward
	bJogBackwards: BOOL;
	/// Jog axis forward
	bJogForward: BOOL;
	/// Slow (starting) speed
	fSlowSpeed: LREAL;
	/// Fast end-speed
	fFastSpeed: LREAL;
	/// Time for ramp from slow to fast speed 
	tAccTime: TIME;
END_STRUCT
END_TYPE

// ---- POUs/Components/AxisDriver/Structures/ST_AxisJogParameter.TcDUT
/// Axis jog parameter strucure
TYPE ST_AxisJogParameter :
STRUCT
	bJogBackwards: BOOL;
	bJogForward: BOOL;
	fAcceleration: LREAL;
	fDeceleration: LREAL;
	fJerk: LREAL;
	eMode: E_JogMode;
	fPosition: LREAL;
	fVelocity: LREAL;
END_STRUCT
END_TYPE

// ---- POUs/Components/AxisDriver/Structures/ST_AxisMoveAbsParameter.TcDUT
/// Axis move absolute parameter strucure
TYPE ST_AxisMoveAbsParameter EXTENDS ST_AxisMoveParameter :
STRUCT
	fPosition: LREAL;
END_STRUCT
END_TYPE

// ---- POUs/Components/AxisDriver/Structures/ST_AxisMoveAddParameter.TcDUT
/// Axis move additive parameter strucure
TYPE ST_AxisMoveAddParameter EXTENDS ST_AxisMoveParameter :
STRUCT
	/// Distance
	fDistance: LREAL;
END_STRUCT
END_TYPE

// ---- POUs/Components/AxisDriver/Structures/ST_AxisMoveModParameter.TcDUT
/// Axis move modulo parameter strucure
TYPE ST_AxisMoveModParameter EXTENDS ST_AxisMoveParameter :
STRUCT
	fPosition: LREAL;
	eDirection: TC2_MC2.MC_Direction;
END_STRUCT
END_TYPE

// ---- POUs/Components/AxisDriver/Structures/ST_AxisMoveParameter.TcDUT
/// General move parameter strucure
TYPE ST_AxisMoveParameter :
STRUCT
	fVelocity: LREAL;
	fAcceleration: LREAL;
	fDeceleration: LREAL;
	fJerk: LREAL;
	fGap: LREAL;
	eBufferMode: MC_BufferMode := MC_Aborting;
	stOptions: ST_MoveOptions;
END_STRUCT
END_TYPE

// ---- POUs/Components/AxisDriver/Structures/ST_AxisMoveRelParameter.TcDUT
/// Axis move relative parameter strucure
TYPE ST_AxisMoveRelParameter EXTENDS ST_AxisMoveParameter :
STRUCT
	/// Distance
	fDistance: LREAL;
END_STRUCT
END_TYPE

// ---- POUs/Components/AxisDriver/Structures/ST_AxisMoveVelParameter.TcDUT
/// Axis move velocity parameter strucure
TYPE ST_AxisMoveVelParameter EXTENDS ST_AxisMoveParameter :
STRUCT
	eDirection: TC2_MC2.MC_Direction;
END_STRUCT
END_TYPE

// ---- POUs/Components/AxisDriver/Structures/ST_AxisSetPosParameter.TcDUT
/// Parameter set for set axis position
TYPE ST_AxisSetPosParameter :
STRUCT
	/// Position to set
	fPosition: LREAL;
	/// RELATIVE=True, ABSOLUTE=False (Default)
	bMode: BOOL;
	/// Additional set position options
	stOptions: ST_SetPositionOptions;
END_STRUCT
END_TYPE

// ---- POUs/Components/AxisDriver/Structures/ST_AxisStopParameter.TcDUT
TYPE ST_AxisStopParameter :
STRUCT
	fDeceleration: LREAL;
	fJerk: LREAL;
	fGap: LREAL;
	stOptions: ST_MoveOptions;
END_STRUCT
END_TYPE

// ---- POUs/Components/AxisDriver/Structures/ST_HmiAxisManager.TcDUT
TYPE ST_HmiAxisManager :
STRUCT
	// axis selection
	eAxis : E_Axis;
	// enable hmi axis mgr
	bEnableAxisMgr : BOOL;

	// global axis manager
	stAxisManager	: REFERENCE TO ST_AxisManager;
END_STRUCT
END_TYPE

// ---- POUs/Components/Device/Structures/ST_DeviceIn.TcDUT
TYPE ST_DeviceIn :
STRUCT
END_STRUCT
END_TYPE

// ---- POUs/Components/Device/Structures/ST_DeviceIO.TcDUT
TYPE ST_DeviceIO :
STRUCT
	stIn 	AT%I* : ST_DeviceIn;
	stOut	AT%Q* : ST_DeviceOut;
END_STRUCT
END_TYPE

// ---- POUs/Components/Device/Structures/ST_DeviceOut.TcDUT
TYPE ST_DeviceOut :
STRUCT
	bRun	: BOOL; // on, off
	fValue	: LREAL; // override, power, ...
END_STRUCT
END_TYPE

// ---- POUs/Components/FurnaceDriver/Enumeration/E_FurnaceSeq.TcDUT
TYPE E_FurnaceSeq :
(
	eFurnaceSeq_none := 0,
	eFurnaceSeq_Auto,
	eFurnaceSeq_Hand,
	eFurnaceSeq_Tune,
	eFurnaceSeq_off
);
END_TYPE

// ---- POUs/Components/FurnaceDriver/Enumeration/E_HeatingState.TcDUT
TYPE E_HeatingState :
(
	eHeatingState_none := 0,
	eHeatingState_on,
	eHeatingState_off
);
END_TYPE

// ---- POUs/Components/FurnaceDriver/Structures/ST_FurnaceIn.TcDUT
{attribute 'pack_mode' := '0'}
TYPE ST_FurnaceIn :
STRUCT	
	nTemperature				: INT;
	bOverheat					: BOOL;
END_STRUCT
END_TYPE

// ---- POUs/Components/FurnaceDriver/Structures/ST_FurnaceIO.TcDUT
/// Turck RFID IO structure.
TYPE ST_FurnaceIO :
STRUCT
	
	/// Data to device.           
	stOut		AT%Q*		: ST_FurnaceOut;
	
	/// Data from device.
	stIn		AT%I*		: ST_FurnaceIn;
	
END_STRUCT
END_TYPE

// ---- POUs/Components/FurnaceDriver/Structures/ST_FurnaceOut.TcDUT
{attribute 'pack_mode' := '0'}
TYPE ST_FurnaceOut :
STRUCT
	bPWMSignal					: BOOL;
END_STRUCT
END_TYPE

// ---- POUs/Components/_Enumerations/E_ComponentState.TcDUT
/// Enumeration of all possible (sub) component states
TYPE E_ComponentState :
(
	/// Component state not set
	eComponentState_none := 0,
	/// Component is resetting
	eComponentState_resetting,
	/// Component is ready
	eComponentState_ready,
	/// Component is running
	eComponentState_running,
	/// Component has error
	eComponentState_error,
	/// Component has warning
	eComponentState_warning,
	/// Component has info
	eComponentState_info
);
END_TYPE

// ---- POUs/Components/_Enumerations/E_Component.TcDUT
/// Enumeration of all plant components
TYPE E_Component :
(
	/// component not set
	eComponent_none := 0,

	/// component max index (keep @ last)
	eComponent_nMaxIdx
);
END_TYPE

// ---- POUs/Components/_Enumerations/E_ComponentType.TcDUT
{attribute 'qualified_only'}
{attribute 'strict'}
TYPE E_ComponentType :
(
	eComponentType_driver,
	eComponentType_axis,
	eComponentType_stateMachine,
	eComponentType_station,
	eComponentType_handler,
	eComponentType_Furnace
);
END_TYPE

// ---- POUs/Components/_Structures/ST_Coordinate.TcDUT
TYPE ST_Coordinate :
STRUCT
fX : REAL;
fY : REAL;
fZ : REAL;
END_STRUCT
END_TYPE

// ---- POUs/Components/_Structures/ST_Curve.TcDUT
TYPE ST_Curve :
STRUCT
	stCurve	: ARRAY[0..0, 0..100] OF ST_Point;
	stColor	: ARRAY[0..0] OF ST_HMI_COLOR_STRING;
END_STRUCT
END_TYPE

// ---- POUs/Components/_Structures/ST_Point.TcDUT
TYPE ST_Point :
STRUCT
	x	: LREAL;
	y	: LREAL;	
END_STRUCT
END_TYPE

// ---- POUs/Components/_Structures/ST_3DPoint.TcDUT
TYPE ST_3DPoint :
STRUCT
	x	: LREAL;
	y	: LREAL;
	z	: LREAL;
END_STRUCT
END_TYPE

// ---- POUs/HMI/Provider/HwHmi/Structures/+P10A_Pult/ST_P10A_Pult_IN.TcDUT
TYPE ST_P10A_Pult_IN :
STRUCT
	bUmlegen	: BOOL; // Umlegen; DT-WH, 2FDI-NO; P10A-51SJ5
	bAufstellen	: BOOL; // Aufstellen; DT-WH, 2FDI-NO; P10A-51SJ7
	bHakenpos	: BOOL; // Hakenposition Anfahren; LDT-BU, 2FDI-NO, 1DO; P10A-51SJ3
	bRichtungL	: BOOL; // Wickelrichtung Links; LDT-WH, 1DI-NO, 1DO; P10A-21SJ1
	bRichtungR	: BOOL; // Wickelrichtung Rechts; LDT-WH, 1DI-NO, 1DO; P10A-21SJ2
	bJogP		: BOOL; // Tippen Vor; DT-WH, 2FDI-NO; P10A-52SJ1
	bJogN		: BOOL; // Tippen Zurück; DT-BK, 2FDI-NO; P10A-52SJ3
END_STRUCT
END_TYPE

// ---- POUs/HMI/Provider/HwHmi/Structures/+P10A_Pult/ST_P10A_Pult_OUT.TcDUT
TYPE ST_P10A_Pult_OUT :
STRUCT
	bLedHakenpos	: BOOL; // Hakenposition Anfahren; LDT-BU, 2FDI-NO, 1DO; P10A-51SJ3
	bLedRichtungL	: BOOL; // Richtung Links; LDT-WH, 1DI-NO, 1DO; P10A-21SJ1
	bLedRichtungR	: BOOL; // Richtung Rechts; LDT-WH, 1DI-NO, 1DO; P10A-21SJ2
END_STRUCT
END_TYPE

// ---- POUs/HMI/Provider/HwHmi/Structures/+P50A_Haupt/ST_P50A_Haupt_IN.TcDUT
TYPE ST_P50A_Haupt_IN :
STRUCT
	bDoorOpn		: BOOL;	// Schutztüren Entriegeln, LDT-WH, 1DI-NO, 1DO, BMK: +P50A-21SJ5
	nOverride		: INT;	// Zustellung Geschwindigkeit, Poti Analog, BMK: +P50A-41SG1
 	bVorwHaerten	: BOOL;	// Vorwahl Härte-Generator, LDT-WH, 1DI-NO, 1DO, BMK: +P50A-22SJ1
	bVorwAnlassen	: BOOL;	// Vorwahl Anlass-Generator, LDT-WH, 1DI-NO, 1DO, BMK: +P50A-22SJ2
	bOnOffPolieren	: BOOL;	// Polierstation Start/Stopp, LDT-WH, 1DI-NO, 1DO, BMK: +P50A-22SJ3
	bSpOnOffS1		: BOOL;	// Spindel S1 Start/Stopp, LDT-WH, 1DI-NO, 1DO, BMK: +P50A-22SJ5
	bSpOnOffS2		: BOOL;	// Spindel S2 Start/Stopp, LDT-WH, 1DI-NO, 1DO, BMK: +P50A-23SJ1
	bSpOnOffS3		: BOOL;	// Spindel S3 Start/Stopp, LDT-WH, 1DI-NO, 1DO, BMK: +P50A-23SJ5
	bAutoOn			: BOOL;	// Automatik Ein, LDT-GN, 1DI-NO, 1DO, BMK: +P50A-21SJ2
	
	bDoorCls		: BOOL;	// Schutztüren Verriegeln, LDT-WH, 1DI-NO, 1DO, BMK: +P50A-21SJ6
	bSchlScheiZust	: BOOL;	// Schleifscheiben Zustellen, DT-WH, 1DI-NO, BMK: +P50A-21SJ7
	bZustOnOffPol	: BOOL;	// Polierstation Zustellung, LDT-WH, 1DI-NO, 1DO, BMK: +P50A-22SJ4
	bZustOnOffS1	: BOOL;	// Spindel S1 Zustellung, LDT-WH, 1DI-NO, 1DO, BMK: +P50A-22SJ6
	bZustOnOffS2	: BOOL;	// Spindel S2 Zustellung, LDT-WH, 1DI-NO, 1DO, BMK: +P50A-23SJ2
	bZustOnOffS3	: BOOL;	// Spindel S3 Zustellung, LDT-WH, 1DI-NO, 1DO, BMK: +P50A-23SJ6
	bAutoOff		: BOOL;	// Automatik Aus, DT-RD, 1DI-NO, BMK: +P50A-21SJ3
	
	bSchlScheiWegst	: BOOL;	// Schleifscheiben Wegstellen, DT-WH, 1DI-NO, BMK: +P50A-21SJ8
	bEnAutoKorrS1	: BOOL;	// Spindel S1 Autokorrektur Ein/Aus, LDT-WH, 1DI-NO, 1DO, BMK: +P50A-22SJ7
	bEnAutoKorrS2	: BOOL;	// Spindel S2 Autokorrektur Ein/Aus, LDT-WH, 1DI-NO, 1DO, BMK: +P50A-23SJ3
	bEnAutoKorrS3	: BOOL;	// Spindel S3 Autokorrektur Ein/Aus, LDT-WH, 1DI-NO, 1DO, BMK: +P50A-23SJ7
	bEsQuit			: BOOL;	// Not-Halt Quittieren, LDT-BU, 1DI-NO, 1DO, BMK: +P50A-21SJ1
END_STRUCT
END_TYPE

// ---- POUs/HMI/Provider/HwHmi/Structures/+P50A_Haupt/ST_P50A_Haupt_OUT.TcDUT
TYPE ST_P50A_Haupt_OUT :
STRUCT
	bLedDoorOpn			: BOOL;	// Schutztüren Entriegeln, LDT-WH, 1DI-NO, 1DO, BMK: +P50A-21SJ5
 	bLedVorwHaerten		: BOOL;	// Vorwahl Härte-Generator, LDT-WH, 1DI-NO, 1DO, BMK: +P50A-22SJ1
	bLedVorwAnlassen	: BOOL;	// Vorwahl Anlass-Generator, LDT-WH, 1DI-NO, 1DO, BMK: +P50A-22SJ2
	bLedPolieren		: BOOL;	// Polierstation Start/Stopp, LDT-WH, 1DI-NO, 1DO, BMK: +P50A-22SJ3
	bLedSpS1			: BOOL;	// Spindel S1 Start/Stopp, LDT-WH, 1DI-NO, 1DO, BMK: +P50A-22SJ5
	bLedSpS2			: BOOL;	// Spindel S2 Start/Stopp, LDT-WH, 1DI-NO, 1DO, BMK: +P50A-23SJ1
	bLedSpS3			: BOOL;	// Spindel S3 Start/Stopp, LDT-WH, 1DI-NO, 1DO, BMK: +P50A-23SJ5
	bLedAutoOn			: BOOL;	// Automatik Ein, LDT-GN, 1DI-NO, 1DO, BMK: +P50A-21SJ2

	bLedDoorCls			: BOOL;	// Schutztüren Verriegeln, LDT-WH, 1DI-NO, 1DO, BMK: +P50A-21SJ6
	bLedHaerteGen		: BOOL;	// Härte-Generator Status, LM-GN, 1DO, BMK: +P50A-32PF2
	bLedAnlassGen		: BOOL;	// Anlss-Generator Status, LM-GN, 1DO, BMK: +P50A-32PF4
	bLedZustPolieren	: BOOL;	// Polierstation Zustellung, LDT-WH, 1DI-NO, 1DO, BMK: +P50A-22SJ4
	bLedZustS1			: BOOL;	// Spindel S1 Zustellung, LDT-WH, 1DI-NO, 1DO, BMK: +P50A-22SJ6
	bLedZustS2			: BOOL;	// Spindel S2 Zustellung, LDT-WH, 1DI-NO, 1DO, BMK: +P50A-23SJ2
	bLedZustS3			: BOOL;	// Spindel S3 Zustellung, LDT-WH, 1DI-NO, 1DO, BMK: +P50A-23SJ6	

	bLedEnAutoKorrS1	: BOOL;	// Spindel S1 Autokorrektur Ein/Aus, LDT-WH, 1DI-NO, 1DO, BMK: +P50A-22SJ7
	bLedEnAutoKorrS2	: BOOL;	// Spindel S2 Autokorrektur Ein/Aus, LDT-WH, 1DI-NO, 1DO, BMK: +P50A-23SJ3
	bLedEnAutoKorrS3	: BOOL;	// Spindel S3 Autokorrektur Ein/Aus, LDT-WH, 1DI-NO, 1DO, BMK: +P50A-23SJ7
	bLedQuit			: BOOL;	// Not-Halt Quittieren, LDT-BU, 1DI-NO, 1DO, BMK: +P50A-21SJ1

END_STRUCT
END_TYPE

// ---- POUs/HMI/Provider/HwHmi/Structures/+P51A_EuchnerHandBedien/ST_P51A_EuchnerHandB_IN.TcDUT
TYPE ST_P51A_EuchnerHandB_IN : //EXTENDS ST_PxAB_SxHandAsBs_IN :
STRUCT
	bSelect01 : BOOL;
	bSelect02 : BOOL;
	bSelect03 : BOOL;
	bSelect04 : BOOL;
	bSelect05 : BOOL;
	bSelect06 : BOOL;
	
	bJog : BOOL;
	bDistance : BOOL;
	bReset : BOOL;
	bAlt : BOOL;
	
	bUp : BOOL;
	bDown : BOOL;
	bLeft : BOOL;
	bRight : BOOL;
END_STRUCT
END_TYPE

// ---- POUs/HMI/Provider/HwHmi/Structures/+P51A_EuchnerHandBedien/ST_P51A_EuchnerHandB_OUT.TcDUT
TYPE ST_P51A_EuchnerHandB_OUT EXTENDS ST_PxAB_SxHandAsBs_OUT:
STRUCT
	bLedSelect01 : BOOL;
	bLedSelect02 : BOOL;
	bLedSelect03 : BOOL;
	bLedSelect04 : BOOL;
	bLedSelect05 : BOOL;
	bLedSelect06 : BOOL;
	 
